(* CODESYS project AxisInterface0.0.1.32.library
   Company: Beckhoff Automation
   DefaultNamespace: BATW
   Version: 0.0.1.32
   Placeholder: AxisInterface
   Author: BATW
   Description: AxisInterface is used to control NC Axis
   Title: AxisInterface

Project tree, tasks and I/O mapping:
  libraries: BATW_Base, * (Beckhoff Automation); Common Behaviour Model, * (3S - Smart Software Solutions GmbH); Tc2_Math, * (Beckhoff Automation GmbH); Tc2_MC2, * (Beckhoff Automation GmbH); Tc2_MC2_Camming, * (Beckhoff Automation GmbH); Tc2_MC2_FlyingSaw, * (Beckhoff Automation GmbH); Tc2_Standard, * (Beckhoff Automation GmbH); Tc2_System, * (Beckhoff Automation GmbH); Tc2_Utilities, * (Beckhoff Automation GmbH); Tc3_JsonXml, * (Beckhoff Automation GmbH); Tc3_MC2_AdvancedHoming, * (Beckhoff Automation GmbH); Tc3_Module, * (Beckhoff Automation GmbH)
  AxisInterface/
    DUT/
      AdvancedHoming/
        data type E_HomingActionType
        data type ST_AdvancedHoming_Parameter
        data type ST_HomingCommand
        data type ST_HomingLimitation
        data type ST_PositionBiasParameter
        data type ST_StepFuncParameter
        data type ST_VelocityParameter
      Axis_Control/
        data type E_PositionType
        data type ST_AXIS_ADMINISTRATION
        data type ST_AXIS_CTRL
        data type ST_AXIS_POSITION
        data type ST_AXIS_SETUP_MODE
        data type ST_AXIS_SYNCHRONISATION
        data type ST_AXIS_SyncPhase
        data type ST_AXIS_SyncProfile
        data type ST_AXIS_SyncVel
        data type ST_AXIS_TORQUE
        data type ST_AXIS_VELOCITY
      Axis_Mode/
        data type E_AXIS_MODE
        data type E_HomingMode
        data type E_StartMode
        data type ST_AXIS_MODE_BITS
        data type U_AXIS_MODE
      Axis_Parameter/
        data type E_OS_Type
        data type ST_AXIS_Parameter
        data type ST_Backlash_Ctrl
        data type ST_Backlash_Status
        data type ST_PositionBias_Ctrl
      Axis_Status/
        data type ST_AXIS_ADMIN_STATUS
        data type ST_AXIS_DIAGNOSIS
        data type ST_AXIS_POS_STATUS
        data type ST_AXIS_SETUP_MODE_STATUS
        data type ST_AXIS_STATUS
        data type ST_AXIS_SYNC_STATUS
        data type ST_AXIS_VEL_STATUS
      CAM/
        data type E_CamID
        data type E_CamTableRef
        data type ST_CamTable
      data type E_AxisDirection
      data type E_MethodStatus_Basic
      data type E_NCI_Status
    GVL/
      global variables AxisInterface_Parameters
      global variables GVL_Motion
    LIB/
      AxisControl/
        program AxisInterface_Type01 [ST]
        function block FB_AdvancedHoming [ST]: M_ClearAllState, M_ClearSignal, M_SetBusy, M_SetDone, M_SetError, M_DogAbs, M_DogDetection, M_LimitDetection, M_LimitFind, M_MoveAbs, M_PulseDetection, M_PulseFind, M_AbortHoming, M_FinishHoming, M_HomeDirect, M_KeepPosBias, A_ActionTrigger, A_CyclicUpdate, M_CheckSignalConnected, M_SelectPreDefinedMode, M_SetUserDefinedMode
        function block FB_AxisControl [ST]: ClearAxisStatusBits, PowerOFF, PowerOn, ReleaseStopAxis, Reset, SetAxisDirction, StopAxis, A00_ModeAB, A01_ModeAH, A02_ModeAdvHoming, A02_ModeHoming, A03_ModePosAbs, A04_ModePosRel, A05_ModePosAdd, A06_ModeVel, A07_ModeSyncPhase, A08_ModeSyncVel, A09_ModeSyncCam, A10_ModeSyncProfile, A11_ModeTorque, A12_ModeFlexProfile, A13_ModeStopping, A14_ModeCoordinated, A15_ModeInterrupted, A16_ModeExternalFB, A17_ModeCyclicPosition, A18_ModeCyclicVelocity, A19_ModeCyclicTorque, A80_AxisParaHandle, A90_Cyclic, M_InitExtension
        function block MC_MoveAbsolute_Continue [ST]
        function block MC_MoveVelocity_Continue [ST]
  Basic Function/
    data type E_JsonHandlerAction
    function block FB_Json_Converter [ST]: JsonStrToObj, ObjToJsonStr
    function block FB_JsonHandler [ST]: CleanupAction, CyclicAction, StartAction, A_CyclicUpdate
  CorrugatedPrint/
    Feeder/
      function F_Poly7_MinTime [ST]
      function F_SolvePoly7Coefficients [ST]
      function block FB_CorrugatedLiftingCalculate [ST]: CleanupAction, CyclicAction, StartAction
      function block FB_CorrugatedWheelThreadCalculate [ST]: CyclicAction, StartAction
  program Main [ST]
*)

// AxisInterface/DUT/AdvancedHoming/E_HomingActionType
{attribute 'qualified_only'}
{attribute 'strict'}
(*
AdvancedHoming Function Type
1.Step Function / Finalizing Function
2.Ref Signal =Limit / Dog / Index
*)
TYPE E_HomingActionType :
(
	(*---Step Function---*)
	Limit_Detection 	:= 0,
	Limit_Abs			:= 1,
	Dog_Detection 		:= 4,
	Dog_Abs				:= 5,
	Index_Detection		:= 6,
	Index_Abs			:= 7,
	(*---Finalizing Function---*)
	HomeDirect			:= 8,
	FinishHoming		:= 9,
	(*---Parameter Setting Step---*)
	ParameterSetting	:=10,
	(*---Abs Motor move to Home---*)
	MoveAbs := 11
);
END_TYPE

// AxisInterface/DUT/AdvancedHoming/ST_AdvancedHoming_Parameter
TYPE ST_AdvancedHoming_Parameter :
STRUCT
	uiCommandNum			:UINT;					//Command List Number
	MovePara_Fast			:ST_VelocityParameter;	//High Speed
	MovePara_Slow			:ST_VelocityParameter;	//Low Speed
	bRefNegLimitSignal		:BOOL;					//Decide the LimitFind Ref Switch(Pos/Neg)
	stHomingCommand			:ARRAY[0..udiMAX_COMMAND_NUM-1] OF ST_HomingCommand;//Command List for Executing Adv Homing
END_STRUCT
END_TYPE

// AxisInterface/DUT/AdvancedHoming/ST_HomingCommand
TYPE ST_HomingCommand :
STRUCT
	eHome_ActionType		:E_HomingActionType;	//AdvancedHoming Function Type
	bSlowVelo				:BOOL;					//True, if Use Low Speed
	stStepFuncParameter		:ST_StepFuncParameter;	//AdvHoming Function Parameter
END_STRUCT
END_TYPE

// AxisInterface/DUT/AdvancedHoming/ST_HomingLimitation
TYPE ST_HomingLimitation :
STRUCT
	TimeLimit		:TIME:=T#0S;
	DistanceLimit	:LREAL:=0;
	TorqueLimit		:LREAL:=0;
END_STRUCT
END_TYPE

// AxisInterface/DUT/AdvancedHoming/ST_PositionBiasParameter
TYPE ST_PositionBiasParameter :
    STRUCT
        bSetPostionBias : BOOL;          //True, then Set Position Bias when Homing end.
        bModuloMode     : BOOL := FALSE; //True: Modulo Bias
    END_STRUCT
END_TYPE

// AxisInterface/DUT/AdvancedHoming/ST_StepFuncParameter
TYPE ST_StepFuncParameter :
STRUCT
	eHome_Direction			:MC_Home_Direction;		//Homing Starting Direction
	eSwitch_Mode			:MC_Switch_Mode;		//Switch Reaction Type
	MovePara				:ST_VelocityParameter;	//Movement Speed,this value should be set by Low/High Speed before Executing Homing Command List
	stHomingLimitation		:ST_HomingLimitation;	//Motion Limitation while searching
END_STRUCT
END_TYPE

// AxisInterface/DUT/AdvancedHoming/ST_VelocityParameter
TYPE ST_VelocityParameter :
STRUCT
	Velocity :LREAL;
	Acc :LREAL;
	Dec : LREAL;
	Jerk: LREAL;
END_STRUCT
END_TYPE

// AxisInterface/DUT/Axis_Control/E_PositionType
{attribute 'qualified_only'}
{attribute 'strict'}
TYPE E_PositionType :
(
	Linear := 0,
	Modulo
);
END_TYPE

// AxisInterface/DUT/Axis_Control/ST_AXIS_ADMINISTRATION
TYPE ST_AXIS_ADMINISTRATION :
    STRUCT
        Axis             : AXIS_REF;    // The reference to this Axis
        _OpMode          : U_AXIS_MODE; // Selection of the operating mode
        ClearError       : BOOL;        // Clear axis error with MC_Reset()
        StopDeceleration : LREAL :=100; // 
        PositionType     : E_PositionType;
        CommandDoneType  : BOOL; //True : real position arrived ;
        stBacklashCtrl   : ST_Backlash_Ctrl;

    END_STRUCT
END_TYPE

// AxisInterface/DUT/Axis_Control/ST_AXIS_CTRL
TYPE ST_AXIS_CTRL :
    STRUCT
        Admin      :ST_AXIS_ADMINISTRATION;  // Administration of the Axis
        PosMode    :ST_AXIS_POSITION;        // Operating mode positioning (absolute, rel, additive)
        VelMode    :ST_AXIS_VELOCITY;        // Operation mode velocity control
        SyncMode   :ST_AXIS_SYNCHRONISATION; // Operation mode synchronisation(phase, vel and cam)
        TorqueMode :ST_AXIS_TORQUE;          // Operation mode / force control
        SetupMode  :ST_AXIS_SETUP_MODE;      // Jog / Homing functionality
		//CoordinatedMode:ST_AXIS_Coordinated; // Operation mode Coordinated control (NCI)
    END_STRUCT
END_TYPE

// AxisInterface/DUT/Axis_Control/ST_AXIS_POSITION
// ST_AXIS_POSITION is a structure that contains the parameters needed when operating in position mode(ABS\REL).
TYPE
    ST_AXIS_POSITION :
    STRUCT
        Position : LREAL;      // The target position value in absolute mode.
        Distance : LREAL;      // The target distance value in relative mode.
        Velocity : LREAL;      // The velocity max value in the position motion.
        Acc : LREAL;           // The accelation max value in the position motion.
        Dec : LREAL;           // The decelation max value in the position motion.
        Jerk : LREAL;          // The jerk max value in the position motion.
        ContinueActive : BOOL; // True : Target command can be change while the motion still running.
    END_STRUCT
END_TYPE

// AxisInterface/DUT/Axis_Control/ST_AXIS_SETUP_MODE
TYPE ST_AXIS_SETUP_MODE :
STRUCT
	eHomingMode			:E_HomingMode;
	FastVelo			:ST_VelocityParameter;
	SlowVelo			:ST_VelocityParameter;
	FastLimitation		:ST_HomingLimitation;//Motion Limitation while Fast Searching
	SlowLimitation		:ST_HomingLimitation;//Motion Limitation while Slow Searching
	lrOffset			:LREAL;//Distance by which the axis moves away from the current position.
	lrSetPosition		:LREAL;//Position value to which the axis position is set to.
	stPosBiasParameter	:ST_PositionBiasParameter;
	
	bHomeSignal :BOOL;
	bPosLimitSignal :BOOL;
	bNegimitSignal :BOOL;
END_STRUCT
END_TYPE

// AxisInterface/DUT/Axis_Control/ST_AXIS_SYNCHRONISATION
TYPE ST_AXIS_SYNCHRONISATION :
STRUCT
	SyncVel :ST_AXIS_SyncVel;
	SyncPhase: ST_AXIS_SyncPhase;
	SyncProfile: ST_AXIS_SyncProfile;
END_STRUCT
END_TYPE

// AxisInterface/DUT/Axis_Control/ST_AXIS_SyncPhase
TYPE
    ST_AXIS_SyncPhase :
    STRUCT
        Master           : AXIS_REF;
        OutputRevolution : LREAL;
        InputRevolution  : UINT;
		MasterSyncPos : LREAL;
		SlaveSyncPos : LREAL;
		MaxAcceleration :LREAL;
		MaxDeceleration : LREAL;
		MaxJerk : LREAL;
		MaxVelocity :LREAL;
		
    //	StartMode        : E_StartMode;

    //  PhaseOffset      : LREAL;

    //  PhaseOffsetVel   : LREAL; // The velocity is used to phasing shift

    //  PhaseOffsetAcc   : LREAL; // The accelation is used to phasing shift

      SyncVelocity     : LREAL; // The velocity is the master axis and slave axis velocity diff in sync process

      SyncAcceleration : LREAL; // The acceleration is the master axis and slace axis acceleration diff in sync process
    END_STRUCT
END_TYPE

// AxisInterface/DUT/Axis_Control/ST_AXIS_SyncProfile
TYPE
    ST_AXIS_SyncProfile :
    STRUCT
        CamProfile    : ARRAY[1..4] OF MC_CAM_REF;
        MasterAxis    : AXIS_REF;
        ProfileNum    : UDINT; // Currently, only profiles 1 to 4 are supported (a total of 4 profiles).
        SyncType      : MC_StartMode;
        Periodic      : BOOL;
        MasterOffset  : LREAL; // Offset for the Master CamIn position, with the unit based on the NC configuration.
        SlaveOffset   : LREAL; // Offset for the Slace CamIn position, wtih the unit based on the NC configuration.
        MasterScaling : LREAL; // Master Axis position data scaling factor, init:1.0
        SlaveScaling  : LREAL; // Slave Axis position data scaling factor, init:1.0
    END_STRUCT
END_TYPE

// AxisInterface/DUT/Axis_Control/ST_AXIS_SyncVel
TYPE
    ST_AXIS_SyncVel :
    STRUCT
        OutputRevolution : LREAL;
        InputRevolution  : UINT;
        FineAdjust       : LREAL;
        Master           : AXIS_REF;
        Acceleration     : LREAL;
        Deceleration     : LREAL;
        Jerk             : LREAL;
    END_STRUCT
END_TYPE

// AxisInterface/DUT/Axis_Control/ST_AXIS_TORQUE
TYPE ST_AXIS_TORQUE :
STRUCT
END_STRUCT
END_TYPE

// AxisInterface/DUT/Axis_Control/ST_AXIS_VELOCITY
TYPE ST_AXIS_VELOCITY :
STRUCT
	Velocity :LREAL;
	Acc :LREAL;
	Dec : LREAL;
	Jerk: LREAL;
END_STRUCT
END_TYPE

// AxisInterface/DUT/Axis_Mode/E_AXIS_MODE
TYPE E_AXIS_MODE :
    (
        ModeAb             := 0,
        ModeAH             := 1,
        ModeHoming         := 2,
        ModePosAbs         := 4,
        ModePosRel         := 8,
        ModePosAdd         := 16,
        ModeVel            := 32,
        ModeSyncPhase      := 64,
        ModeSyncVel        := 128,
        ModeSyncCam        := 256,
        ModeSyncProfile    := 512,
        ModeTorque         := 1024,
        ModeFlexProfile    := 2048,
        ModeStopping       := 4096,
        ModeCoordinated    := 8192,
        ModeInterrupted    := 16384,
        ModeExternalFB     := 32768,
        ModeCyclicPosition := 65536,
        ModeCyclicVelocity := 131072,
        ModeCyclicTorque   := 262144
    )UDINT;
END_TYPE

// AxisInterface/DUT/Axis_Mode/E_HomingMode
{attribute 'qualified_only'}
{attribute 'strict'}
//CiA402 Homing Mode
(*-----------------

_03  					=> Mode Number
_Pos 					=> Start Direction
_LimitOutterLeftIndex 	=> Final target position
_withLimit				=> Action will reverse when meets limit

-----------------*)
TYPE E_HomingMode :
(
	notDefined									:=0,
                              	
	//Limit Switch plus Index           	
	_01_Neg_LimitOutterRightIndex				:=1,
	_02_Pos_LimitOutterLeftIndex 				:=2,
	
	//Single Transition Home Switch plus Index
	_03_Pos_HomeOutterLeftIndex					:=3,
	_04_Pos_HomeInnerLeftIndex					:=4,
	_05_Neg_HomeOutterRightIndex				:=5,
	_06_Neg_HomeInnerRightIndex					:=6,
	
	//Limited Range Home Switch, Limit Switched and Index
	_07_Pos_HomeOutterLeftIndex_withLimit		:=7,
	_08_Pos_HomeInnerLeftIndex_withLimit		:=8,
	_09_Pos_HomeInnerRightIndex_withLimit		:=9,
	_10_Pos_HomeOutterRightIndex_withLimit		:=10,
	_11_Neg_HomeOutterRightIndex_withLimit		:=11,
	_12_Neg_HomeInnerRightIndex_withLimit		:=12,
	_13_Neg_HomeInnerLeftIndex_withLimit		:=13,
	_14_Neg_HomeOutterLeftIndex_withLimit		:=14,
	
	//----------------------------//
	//Home on Limit Switch
	_17_Neg_LimitOutterRight				:=17,
	_18_Pos_LimitOutterLeft					:=18,
	
	//Single Transition Home Switch
	_19_Pos_HomeOutterLeft					:=19,
	_20_Pos_HomeInnerLeft					:=20,
	_21_Neg_HomeOutterRight					:=21,
	_22_Neg_HomeInnerRight					:=22,
	
	//Two Transition Home Switch and Limit Switches
	_23_Pos_HomeOutterLeft_withLimit		:=23,
	_24_Pos_HomeInnerLeft_withLimit			:=24,
	
	//Two Transition Home Switch, Limit Switches and Index
	_25_Pos_HomeInnerRight_withLimit		:=25,
	_26_Pos_HomeOutterRight_withLimit		:=26,
	_27_Neg_HomeOutterRight_withLimit		:=27,
	_28_Neg_HomeInnerRight_withLimit		:=28,
	_29_Neg_HomeInnerLeft_withLimit			:=29,
	_30_Neg_HomeOutterLeft_withLimit		:=30,

	//Index
	_33_Neg_Index			:=33,
	_34_Pos_Index			:=34,
	                                        	
	//Set to current position               	
	_35_CurrentPosition		:=35,
	
	// Absolute Motor move to home point
	_36_MoveToAbsHomePoint := 36
	//--------------Customized--------------//
	//_36_CurrentPosition_WithBias	:=36
	
	
	
);
END_TYPE

// AxisInterface/DUT/Axis_Mode/E_StartMode
{attribute 'qualified_only'}
{attribute 'strict'}
TYPE E_StartMode :
(
	Absolute := 0, // flying coupling with abs sync only first execution
	Relative :=1, // flying coupling with rel sync only first execution
	Absolute_Rampin, // flying coupling with abs sync every execution
	Relative_Rampin // flying coupling with rel sync ecery execution
);
END_TYPE

// AxisInterface/DUT/Axis_Mode/ST_AXIS_MODE_BITS
TYPE ST_AXIS_MODE_BITS :
    STRUCT
        ModeAH             :BIT;
        ModeHoming         :BIT;
        ModePosAbs         :BIT;
        ModePosRel         :BIT;
        ModePosAdd         :BIT;
        ModeVel            :BIT;
        ModeSyncPhase      :BIT;
        ModeSyncVel        :BIT;
        ModeSyncCam        :BIT;
        ModeSyncProfile    :BIT;
        ModeTorque         :BIT;
        ModeFlexProfile    :BIT;
        ModeStopping       :BIT;
        ModeCoordinated    :BIT;
        ModeInterrupted    :BIT;
        ModeExternalFB     :BIT;
        ModeCyclicPosition :BIT;
        ModeCyclicVelocity :BIT;
        ModeCyclicTorque   :BIT;
    END_STRUCT
END_TYPE

// AxisInterface/DUT/Axis_Mode/U_AXIS_MODE
TYPE U_AXIS_MODE :
UNION
	en : E_AXIS_MODE;
	b: ST_AXIS_MODE_BITS;
END_UNION
END_TYPE

// AxisInterface/DUT/Axis_Parameter/E_OS_Type
{attribute 'qualified_only'}
{attribute 'strict'}
TYPE E_OS_Type :
(
	WinCE 	:= 0,
	Windows := 1
);
END_TYPE

// AxisInterface/DUT/Axis_Parameter/ST_AXIS_Parameter
TYPE ST_AXIS_Parameter :
STRUCT
	(* -----Parameter----- *)
	(* Position Bias *)
	stPositionBias_Ctrl		:ST_PositionBias_Ctrl;
	
	(* Backlash *)
	stBacklash_Ctrl			:ST_Backlash_Ctrl;
	
END_STRUCT
END_TYPE

// AxisInterface/DUT/Axis_Parameter/ST_Backlash_Ctrl
TYPE ST_Backlash_Ctrl :
STRUCT
	bEnable		:BOOL;		//true, enable backlash compensation
	lrRamp		:LREAL:=1;	//Velocity limit for entered backlash compensation. [mm/s]
	lrBacklash	:LREAL:=0;	//Backlash Value
	bIsPosDir	:BOOL:=TRUE;//True, if Backlash compensation for Pos Direction
END_STRUCT
END_TYPE

// AxisInterface/DUT/Axis_Parameter/ST_Backlash_Status
TYPE ST_Backlash_Status :
STRUCT
	lrCurrentBacklash	:LREAL;//Current compensation value [mm].
	
	
END_STRUCT
END_TYPE

// AxisInterface/DUT/Axis_Parameter/ST_PositionBias_Ctrl
TYPE ST_PositionBias_Ctrl :
STRUCT
	lrPosBiasValue	:LREAL;//Position Bias Value 
	bSetPostionBias	:BOOL;//True, then Set Position Bias when Homing end.
	bModuloMode		:BOOL;//True=Modulo Bias
END_STRUCT
END_TYPE

// AxisInterface/DUT/Axis_Status/ST_AXIS_ADMIN_STATUS
TYPE
    ST_AXIS_ADMIN_STATUS :
    STRUCT
        Active             : BOOL;               // True: The drive is actived / PowerOn / Servo On
        CmdDone            : BOOL;               // Last motion command is finished
        _OpModeAck         : E_AXIS_MODE;        // acknowledge of the operation mode
        DriverAddress      : ST_DriveAddress;    // Read Driver Address
        stBacklash_Status  : ST_Backlash_Status; //Backlash Status
        ModeAb             : BIT;                // The axis is in Ab mode.
        ModeAH             : BIT;                // The axis is in AH mode.
        ModeHoming         : BIT;                // The axis is in homing mode.
        ModePosAbs         : BIT;                // The axis is in position absolute mode.
        ModePosRel         : BIT;                // This axis is in position relative mode.
        ModePosAdd         : BIT;                // This axis is in position additive mode.
        ModeVel            : BIT;                // This axis is in velocity control mode.
        ModeSyncPhase      : BIT;                // This axis is in synchronize phase mode.
        ModeSyncVel        : BIT;                // This axis is in synchronize velocity mode.
        ModeSyncCam        : BIT;                // This axis is in synchronize Cam mode.
        ModeSyncProfile    : BIT;                // This axis is in synchronize Cam Profile mode.
        ModeTorque         : BIT;                // This axis is in torque control mode.
        ModeFlexProfile    : BIT;                // This axis is in synchronize Cam-> FlexProfile mode.
        ModeStopping       : BIT;                // This axis is in stopping mode.
        ModeCoordinated    : BIT;                // This axis is in coordinated mode.
        ModeInterrupted    : BIT;                // This axis is in interrupted mode.
        ModeExternalFB     : BIT;                // This axis is using exeternal FB.
        ModeCyclicPosition : BIT;                // This axis is in cyclic Position control mode.
        ModeCyclicVelocity : BIT;                // This axis is in cyclic Velocity control mode.
        ModeCyclicTorque   : BIT;                // This axis is in cyclic torque control mode.
    END_STRUCT
END_TYPE

// AxisInterface/DUT/Axis_Status/ST_AXIS_DIAGNOSIS
TYPE ST_AXIS_DIAGNOSIS :
STRUCT
	Warning :BOOL := FALSE;
	Error : BOOL:=FALSE;
	ErrorID : UDINT;
	ErrorMsg : T_MaxString;
END_STRUCT
END_TYPE

// AxisInterface/DUT/Axis_Status/ST_AXIS_POS_STATUS
TYPE ST_AXIS_POS_STATUS :
STRUCT
END_STRUCT
END_TYPE

// AxisInterface/DUT/Axis_Status/ST_AXIS_SETUP_MODE_STATUS
TYPE ST_AXIS_SETUP_MODE_STATUS :
STRUCT
END_STRUCT
END_TYPE

// AxisInterface/DUT/Axis_Status/ST_AXIS_STATUS
TYPE ST_AXIS_STATUS :
    STRUCT
        Admin     :ST_AXIS_ADMIN_STATUS; 
        Diag      :ST_AXIS_DIAGNOSIS;
        PosMode   :ST_AXIS_POS_STATUS;
        VelMode   :ST_AXIS_VEL_STATUS;
        SyncMode  :ST_AXIS_SYNC_STATUS;
        SetupMode :ST_AXIS_SETUP_MODE_STATUS;
    END_STRUCT
END_TYPE

// AxisInterface/DUT/Axis_Status/ST_AXIS_SYNC_STATUS
TYPE
    ST_AXIS_SYNC_STATUS :
    STRUCT
        ModuleGap : LREAL;
    END_STRUCT
END_TYPE

// AxisInterface/DUT/Axis_Status/ST_AXIS_VEL_STATUS
TYPE ST_AXIS_VEL_STATUS :
STRUCT
END_STRUCT
END_TYPE

// AxisInterface/DUT/CAM/E_CamID
{attribute 'qualified_only'}
{attribute 'strict'}
TYPE E_CamID :
(
	Undefined := 0,
	Cam1 :=1,
	Cam2 :=2,
	Cam3 :=3,
	Cam4 :=4
)UDINT;
END_TYPE

// AxisInterface/DUT/CAM/E_CamTableRef
{attribute 'qualified_only'}
{attribute 'strict'}
TYPE
    E_CamTableRef :
    (
        Undefined := 0,
        CamTable_01 := 1,
        CamTable_02 := 2,
        CamTable_03 := 3,
        CamTable_04 := 4
    );
END_TYPE

// AxisInterface/DUT/CAM/ST_CamTable
TYPE
    ST_CamTable :
    STRUCT
        CamTable_01 : MC_CAM_REF;
        CamTable_02 : MC_CAM_REF;
        CamTable_03 : MC_CAM_REF;
        CamTable_04 : MC_CAM_REF;
    END_STRUCT
END_TYPE

// AxisInterface/DUT/E_AxisDirection
TYPE E_AxisDirection :
(
	Locked := 0,
	OnlyPositive,
	OnlyNegative,
	Both
)UINT;
END_TYPE

// AxisInterface/DUT/E_MethodStatus_Basic
// Declare the basic level that a method typically goes through, based on PLC Open OOP guidelines.
{attribute 'strict'}
TYPE E_MethodStatus_Basic :
(
	STATE_DORMANT := 0, // In dormant state, do nothing and just wait for the start command.
	STATE_EXECUTING, 	// In executing state, the state will do something that you coded
	STATE_ABORTING, 	// In aborting state, stop all ongoing commands.
	STATE_DONE, 		// In done state, waitting the reset command or execute signal off
	STATE_Aborted, 		// In aborted state, method is frozen wait reset command or execute signal off
	STATE_ERROR,		// In error state, method has been stopped and only can be restart by reset command or execute signal off 
	STATE_RESETTING    	// In resetting state, the state will revert the status to its initial values and clear any error signals.
)UDINT;
END_TYPE

// AxisInterface/DUT/E_NCI_Status
TYPE E_NCI_Status :
(
	NCI_INITFAILED := 0,
	NCI_IDLE,
	NCI_READY,
	NCI_STARTED,
	NCI_SCANNING,
	NCI_RUNNING,
	NCI_STAY_RUNNING,
	NCI_WRITETABLE,
	NCI_SEARCHLINE,
	NCI_END,
	NCI_SINGLESTOP,
	NCI_ABORTING,
	NCI_ABORTED,
	NCI_FAULT,
	NCI_RESET,
	NCI_STOP,
	NCI_WAITFUNC,
	NCI_FLUSHBUFFERS
)UDINT;
END_TYPE

// Basic Function/E_JsonHandlerAction
{attribute 'qualified_only'}
{attribute 'strict'}
TYPE E_JsonHandlerAction :
(
	READ 	:= 0,
	WRITE	:= 1
);
END_TYPE

// AxisInterface/GVL/AxisInterface_Parameters
VAR_GLOBAL CONSTANT
    uiMAX_AXIS_INDEX   		: UINT := 10;  // Maximum number of servos in the system.
    uiMAX_AXIS_NUMBER  		: UINT := 4;   // Actual number of servos in the system.
    udiMAX_COMMAND_NUM 		: UDINT := 10; //Maximum number of Advanced Homing command 
	eOsType			   		: E_OS_Type:=E_OS_Type.Windows;//OS Type,decide deafaut Axis Para file folder
	sAxisParaFolderPath  	: T_MaxString:='';//Axis Parameter File Folder ,example: 'C:\TwinCAT\3.1\Boot'
END_VAR

// AxisInterface/GVL/GVL_Motion
VAR_GLOBAL
    arAxisCtrl_gb     :ARRAY[1..uiMAX_AXIS_INDEX] OF ST_AXIS_CTRL;
    arAxisStatus_gb   :ARRAY[1..uiMAX_AXIS_INDEX] OF ST_AXIS_STATUS;
END_VAR
VAR_GLOBAL PERSISTENT
	arAxisPara_gb	  :ARRAY[1..uiMAX_AXIS_INDEX] OF ST_AXIS_Parameter;
	//arAxisBias_gb     		:ARRAY[1..uiMAX_AXIS_INDEX] OF LREAL;
END_VAR

// AxisInterface/LIB/AxisControl/AxisInterface_Type01
PROGRAM AxisInterface_Type01
VAR
    {attribute 'hide'}
    uiLoop :UINT; // For loop index
    {attribute 'hide'}
    fbAxis :ARRAY[1..uiMAX_AXIS_NUMBER] OF FB_AxisControl; // IMPLEMENTS axis control fb
	uiIndex : UINT;
	
	bDogSignal_Simu:BOOL;
	bPosLimitSiganl_Simu:BOOL;
	bNegLimitSignal_Simu:BOOL;
	
END_VAR

VAR CONSTANT
END_VAR

//============================================//
// Reflash Axis Interface					  //
//============================================//

FOR uiLoop := 1 TO uiMAX_AXIS_NUMBER DO
    fbAxis[uiLoop].M_InitExtension(uiLoop);
    //fbAxis[uiLoop]();
    fbAxis[uiLoop](HomeSensor := arAxisCtrl_gb[uiLoop].SetupMode.bHomeSignal,
                   PosLimit := arAxisCtrl_gb[uiLoop].SetupMode.bPosLimitSignal,
                   NegLimit := arAxisCtrl_gb[uiLoop].SetupMode.bNegimitSignal);
END_FOR

END_PROGRAM

// AxisInterface/LIB/AxisControl/FB_AxisControl
{attribute 'reflection'}
FUNCTION_BLOCK FB_AxisControl
VAR_INPUT
    HomeSensor : BOOL;
    PosLimit   : BOOL;
    NegLimit   : BOOL;

    {attribute 'hide'}
    bThirdPartyDrive : BOOL := TRUE;
END_VAR

VAR_OUTPUT
END_VAR

VAR
    // Control unit
    PowerControl          : Tc2_MC2.MC_Power; // MC_Power, Declare the use of a function block.
    ResetControl          : Tc2_MC2.MC_Reset; // MC_Reset, Declare the use of a function block.
    StopControl           : Tc2_MC2.MC_Stop; // MC_Stop, Declare the use of a function block.
    HaltControl           : Tc2_MC2.MC_Halt; // MC_Halt, Declare the use of a function block.
    JogControl            : Tc2_MC2.MC_Jog; // MC_Jog, Declare the use of a function block.
    HomingControl         : Tc2_MC2.MC_Home; // MC_Home, Declare the use of a function block.
    MoveAbsControl        : Tc2_MC2.MC_MoveAbsolute; // MC_MoveAbsolute, Declare the use of a function block.
    MoveRelControl        : Tc2_MC2.MC_MoveRelative; // MC_MoveRelative, Declare the use of a function block.
    MoveAddControl        : Tc2_MC2.MC_MoveAdditive; // MC_ModeAdditive, Declare the use of a function block.
    MoveModuleControl     : Tc2_MC2.MC_MoveModulo; // MC_MoveModule, Declare the use of a function block.
    MoveVelControl        : Tc2_MC2.MC_MoveVelocity; // MC_MoveVelocitu, Declare the use of a function block.
    MoveVelControl_Ext    : MC_MoveVelocity_Continue; // MC_MoveVelocity_Continue, Declare the use of a function block.
    MoveAbsolute_Ext      : MC_MoveAbsolute_Continue; // MC_MoveAbsolute_Continue, Declare the use of a function block.
    SyncVelControl        : MC_GearInVelo; // MC_GearInVelo, Declare the use of a function block.
    SyncPhaseControl      : MC_GearInPos; // MC_GearInPos, Declare the use of a function block.
    SetPositionControl    : MC_SetPosition; // MC_SetPositionControl, Declare the use of a function block.
    CamSelector           : MC_CamTableSelect; // MC_CamTableSelect, Declare the use of a function block.
    CamInControl          : MC_CamIn; // MC_CamIn, Declare the use of a function block.
    fbAdvancedHoming      : FB_AdvancedHoming; // FB_AdvancedHoming, Declare the use of a function block.
    fbBacklash            : MC_BacklashCompensation;
    PhasingAbsControl     : MC_PhasingAbsolute; // MC_PhasingAbsolute, Declare the use of a function block.
    PhasingRelControl     : MC_PhasingRelative; // MC_PhasingRelative, Declare the use of a function block.
    PhaseOffset_Abs       : LREAL;
    PhaseOffset_Rel       : LREAL;
    PhaseOffsetSuperInpos : MC_MoveSuperImposed;
    SuperInposMode        : E_SuperpositionMode;
    fbWriteNcPara         : MC_WriteParameterPersistent; //Read NC Parameter
    fbReadNcPara          : MC_ReadParameter; //Write NC Parameter
    fbWritePersistent     : FB_WritePersistentData;
    fbAxisParaHandler     : FB_JsonHandler;
    GearOutControl        : MC_GearOut;

    // Axis command 
    AxisPowerON       : BOOL; // True: set mc_power.enable = True
    AllowPositiveMove : BOOL; // True: Allow axis move to positive direction
    AllowNegativeMove : BOOL; // True: Allow axis move to Negative direction
    AxisStop          : BOOL; // True: Set mc_Stop.Execute = true
    AxisStop_Dec      : LREAL := 1000; // mc_Stop's deceleration
    AxisStop_Jerk     : LREAL := 10000; // mc_Stop's jerk
    AxisID            : UDINT;
    //-----Axis Parameter-----//
    //
    bInitializePosBiasDone : BOOL := FALSE;
    bReadAxisPara          : BOOL;
    sTempString            : STRING(255);
    sTempString2           : STRING(255);
    retryTimer             : TON;
    fbWritePersistentdata  : FB_WritePersistentData;
    lrNcCurrentBias        : LREAL;
    lrStoredBias           : LREAL;
    bAxisInitDone          : BOOL := FALSE;
    bAxisDoingInit         : BOOL := FALSE;
    uiAxisInitRetryCount   : UINT;

    //BackLash
    bBacklash_Enable   : BOOL; //true, enable backlash compensation
    lrBacklash_Ramp    : LREAL := 1; //Velocity limit for entered backlash compensation. [mm/s]
    lrBacklash_Value   : LREAL := 0; //Backlash Value
    bBacklash_IsPosDir : BOOL  := TRUE; //True, if Backlash compensation for Pos Direction

    // Cam Table
    CamProfileIndex : UDINT; // Cam Profile number (1~4)
    arCamID         : ARRAY[1..4] OF UDINT; // Store the actual CAM ID

    //A02 advance homing
    SetPosition_Execute       : BOOL;
    SetPosition_Position      : LREAL; // This value will be set to Absoulte position
    advHoming_eHomingMode     : E_HomingMode;
    advHoming_FastVelo        : ST_VelocityParameter;
    advHoming_SlowVelo        : ST_VelocityParameter;
    advHoming_lrOffset        : LREAL; //Distance by which the axis moves away from the current position.
    advHoming_lrSetPosition   : LREAL; //Position value to which the axis position is set to.
    advHoming_StartHoming     : BOOL;
    advHoming_AbortHoming     : BOOL;
    advHoming_ThirdPartyDrive : BOOL;
    {attribute 'is_connected' := 'HomeSensor'}
    advHoming_bDogConnected : BOOL;
    {attribute 'is_connected' := 'PosLimit'}
    advHoming_bPosLimitConnected : BOOL;
    {attribute 'is_connected' := 'NegLimit'}
    advHoming_bNegLimitConnected : BOOL;
    advHoming_PositionBiasPara   : ST_PositionBiasParameter;
	// A03
    PosAbsMode_Execute         : BOOL;
    PosAbsMode_Position        : LREAL;
    PosAbsMode_Velocity        : LREAL;
    PosAbsMode_Acc             : LREAL;
    PosAbsMode_Dec             : LREAL;
    PosAbsMode_Jerk            : LREAL;
    PosAbsMode_Exectue_Modulo  : BOOL;
    PosAbsMode_Position_Modulo : LREAL;
    PosAbsMode_Velocity_Modulo : LREAL;
    PosAbsMode_Acc_Modulo      : LREAL;
    PosAbsMode_Dec_Modulo      : LREAL;
    PosAbsMode_Jerk_Modulo     : LREAL;
	PosAbsMode_Direction : MC_Direction:=MC_Direction.MC_Shortest_Way;
	PosAbsMode_LastPosition : LREAL;
    //A04
    PosRelMode_Execute  : BOOL;
    PosRelMode_Distance : LREAL;
    PosRelMode_Velocity : LREAL;
    PosRelMode_Acc      : LREAL;
    PosRelMode_Dec      : LREAL;
    PosRelMode_Jerk     : LREAL;

    // A06
    VelMode_Velocity : LREAL := 0;
    VelMode_Acc      : LREAL := 10;
    VelMode_Dec      : LREAL := 10;
    VelMode_Jerk     : LREAL := 100;
    VelMode_Dir      : MC_Direction;
    VelMode_Execute  : BOOL;

    //A07 ModeSyncPhase
    SyncPhaseMode_Enable           : BOOL;
    SyncPhaseMode_Master           : REFERENCE TO AXIS_REF;
    SyncPhaseMode_RatioNumerator   : LREAL;
    SyncPhaseMode_RatioDenominator : UINT;
    SyncPhaseMode_MasterSyncPos    : LREAL := 0;
    SyncPhaseMode_SlaveSyncPos     : LREAL := 0;
    SyncPhaseMode_SyncMode         : ST_SyncMode;
    //SyncPhaseMode_MasterStartPos   : LREAL;
    SyncPhaseMode_MaxVelocity       : LREAL := 10;
    SyncPhaseMode_MaxAcc            : LREAL;
    SyncPhaseMode_MaxDec            : LREAL;
    SyncPhaseMode_MaxJerk           : LREAL;
    SyncPhaseMode_RealMasterPos     : LREAL;
    SyncPhaseMode_RealSlavePos      : LREAL;
    SyncPhaseMode_LastMasterSyncPos : LREAL;
    SyncPhaseMode_LastSlaveSyncPos  : LREAL;
    SyncPhaseMode_SyncVelocity      : LREAL;
    SyncPhaseMode_SyncAcceleration  : LREAL;
    //A08 ModeSyncVel
    SyncVelMode_Enable           : BOOL;
    SyncVelMode_Master           : REFERENCE TO AXIS_REF;
    SyncVelMode_GearRatio        : LREAL;
    SyncVelMode_RatioNumerator   : LREAL;
    SyncVelMode_RatioDenominator : UINT;
    SyncVelMode_SyncMode         : ST_SyncMode;
    SyncVelMode_FineAdjust       : LREAL;
    SyncVelMode_Acc              : LREAL;
    SyncVelMode_Dec              : LREAL;
    SyncVelMode_Jerk             : LREAL;

    //A10 ModeSyncProfile
    SyncProfileMode_Master        : REFERENCE TO AXIS_REF;
    SyncProfileMode_ProfileNum    : UDINT;
    SyncProfileMode_SyncType      : MC_StartMode;
    SyncProfileMode_MasterOffset  : LREAL;
    SyncProfileMode_SlaveOffset   : LREAL;
    SyncProfileMode_MasterScaling : LREAL := 1.0;
    SyncProfileMode_SlaveScaling  : LREAL := 1.0;
    SyncProfileMode_Periodic      : BOOL;
    SyncProfileMode_CamID         : MC_CAM_ID;
    SyncProfileOption             : ST_CamInOptions;

    //A17 ModeCyclicPosition
    PosCyclicAbsMode_Execute  : BOOL;
    PosCyclicAbsMode_Position : LREAL;
    PosCyclicAbsMode_Velocity : LREAL;
    PosCyclicAbsMode_Acc      : LREAL;
    PosCyclicAbsMode_Dec      : LREAL;
    PosCyclicAbsMode_Jerk     : LREAL;

    // Action state
    uiModeAb_State                      : UINT; // ModeAb's current state 
    uiModeAH_State                      : UINT; // ModeAH's current state
    uiModeHoming_State                  : UINT; // ModeHoming's current state
    uiModeCoordinatedState              : UINT; // ModeCoordinated current State
    uiModeVelState                      : UINT; // ModeVel's current state
    uiModePosAbsState                   : UINT; // ModePosAbs's current state
    uiModePosRelState                   : UINT; // ModePosRel's current state
    uiModeCyclicPosAbsState             : UINT; // ModePosAbs's current state
    uiModeSyncVelState                  : UINT; // ModeSyncVel's current state
    uiModeSyncPhaseState                : UINT; // ModeSyncPhase's current state
    uiModeSyncProfile                   : UINT; // ModeSyncProfile's current state
    uiModeFlexProfileState              : UINT; // ModeSyncFlexProfile current state
    LastOpMode                          : E_AXIS_MODE; // record last mode
    SyncPhaseMode_SlaveModuleTurns      : LREAL;
    SyncPhaseMode_SlaveModuleRemainder  : LREAL;
    SyncPhaseMode_MasterModuleTurns     : LREAL;
    SyncPhaseMode_MasterModuleRemainder : LREAL;
    SuperInposDistance                  : LREAL;
    AxesGap                             : LREAL;
    LastSuperInposDistance              : LREAL;

    // Read Axis Address
    fbReadAxisAddress : MC_ReadDriveAddress;
    AxesGap2          : LREAL;
    AxesGap3          : LREAL;
	ModuleGap: LREAL;
END_VAR

VAR
    {attribute 'no_copy'}
    AdminCtrl : REFERENCE TO ST_AXIS_ADMINISTRATION; // Reference to arAxisCtrl.admin
    {attribute 'no_copy'}
    PosModeCtrl : REFERENCE TO ST_AXIS_POSITION; // Reference to arAxisCtrl.PosMode
    {attribute 'no_copy'}
    VelModeCtrl : REFERENCE TO ST_AXIS_VELOCITY; // Reference to arAxisCtrl.VelMode
    {attribute 'no_copy'}
    SyncModeCtrl : REFERENCE TO ST_AXIS_SYNCHRONISATION; // Reference to arAxisCtrl SyncMode
    {attribute 'no_copy'}
    TorqueModeCtrl : REFERENCE TO ST_AXIS_TORQUE; // Reference to arAxisCtrl TorqueMode
    {attribute 'no_copy'}
    SetupModeCtrl : REFERENCE TO ST_AXIS_SETUP_MODE; // Reference to arAxisCtrl SetupMode
    {attribute 'no_copy'}
    AdminStatus : REFERENCE TO ST_AXIS_ADMIN_STATUS; // Reference to arAxisStat
    {attribute 'no_copy'}
    DiagStatus : REFERENCE TO ST_AXIS_DIAGNOSIS;
    {attribute 'no_copy'}
    PosModeStatus : REFERENCE TO ST_AXIS_POS_STATUS;
    {attribute 'no_copy'}
    VelModeStatus : REFERENCE TO ST_AXIS_VEL_STATUS;
    {attribute 'no_copy'}
    SyncModeStatus : REFERENCE TO ST_AXIS_SYNC_STATUS;
    {attribute 'no_copy'}
    SetupModeStatus : REFERENCE TO ST_AXIS_SETUP_MODE_STATUS;
    {attribute 'no_copy'}
    //refNcPositionBias : REFERENCE TO LREAL;//Reference to arAxisBias_gb
    {attribute 'no_copy'}
    refAxisPara : REFERENCE TO ST_AXIS_Parameter; //Reference to arAxisPara_gb
END_VAR

IF NOT __ISVALIDREF(AdminCtrl) THEN
    RETURN;
END_IF

// ----------------------------------------------- //
// ----------- Action ---------------------------- //
A00_ModeAB();
A01_ModeAH();
//A02_ModeHoming();
A02_ModeAdvHoming();
A03_ModePosAbs();
A04_ModePosRel();
A05_ModePosAdd();
A06_ModeVel();
A07_ModeSyncPhase();
A08_ModeSyncVel();
A09_ModeSyncCam();
A10_ModeSyncProfile();
A11_ModeTorque();
A12_ModeFlexProfile();
A13_ModeStopping();
A14_ModeCoordinated();
A15_ModeInterrupted();
A16_ModeExternalFB();
A17_ModeCyclicPosition();
A18_ModeCyclicVelocity();
A19_ModeCyclicTorque();

A90_Cyclic();

(* Axis Parameter Read/Write *)
A80_AxisParaHandle();

IF AdminCtrl.Axis.Status.Coupled THEN
    IF (SyncModeCtrl.SyncPhase.Master.NcToPlc.ModuloSetPos - AdminCtrl.Axis.NcToPlc.ModuloSetPos) >= 0 THEN
        ModuleGap := (SyncModeCtrl.SyncPhase.Master.NcToPlc.ModuloSetPos - AdminCtrl.Axis.NcToPlc.ModuloSetPos);
    ELSE
        ModuleGap := 360 + (SyncModeCtrl.SyncPhase.Master.NcToPlc.ModuloSetPos - AdminCtrl.Axis.NcToPlc.ModuloSetPos);
    END_IF
ELSE
    IF (SyncModeCtrl.SyncPhase.Master.NcToPlc.ModuloActPos - AdminCtrl.Axis.NcToPlc.ModuloActPos) >= 0 THEN
        ModuleGap := (SyncModeCtrl.SyncPhase.Master.NcToPlc.ModuloActPos - AdminCtrl.Axis.NcToPlc.ModuloActPos);
    ELSE
        ModuleGap := 360 + (SyncModeCtrl.SyncPhase.Master.NcToPlc.ModuloActPos - AdminCtrl.Axis.NcToPlc.ModuloActPos);
    END_IF
END_IF

SyncModeStatus.ModuleGap := ModuleGap;

METHOD PRIVATE ClearAxisStatusBits
VAR_INPUT
END_VAR
AdminStatus.ModeAb := FALSE;
AdminStatus.ModeAH := FALSE;
AdminStatus.ModeCoordinated := FALSE;
AdminStatus.ModeCyclicPosition := FALSE;
AdminStatus.ModeCyclicTorque := FALSE;
AdminStatus.ModeCyclicVelocity := FALSE;
AdminStatus.ModeExternalFB := FALSE;
AdminStatus.ModeFlexProfile := FALSE;
AdminStatus.ModeHoming := FALSE;
AdminStatus.ModeInterrupted := FALSE;
AdminStatus.ModePosAbs := FALSE;
AdminStatus.ModePosAdd := FALSE;
AdminStatus.ModePosRel := FALSE;
AdminStatus.ModeStopping := FALSE;
AdminStatus.ModeSyncCam := FALSE;
AdminStatus.ModeSyncPhase := FALSE;
AdminStatus.ModeSyncProfile := FALSE;
AdminStatus.ModeSyncVel := FALSE;
AdminStatus.ModeTorque := FALSE;
AdminStatus.ModeVel := FALSE;
END_METHOD

METHOD PRIVATE PowerOFF
VAR_INPUT
END_VAR
IF NOT PowerControl.Status THEN
    RETURN;
END_IF

AllowPositiveMove := FALSE;
AllowNegativeMove := FALSE;
AxisPowerON := FALSE;
END_METHOD

METHOD PRIVATE PowerOn
VAR_INPUT
    Direction :E_AxisDirection; // set the movable directions of the Axis.
END_VAR
VAR CONSTANT
	STATE_CHECK_AXISPOWER : UINT:=0;
	STATE_SET_POWER_PARA : UINT:=1;
END_VAR
IF PowerControl.Status THEN
	RETURN;
END_IF

SetAxisDirction(Direction:= Direction);

AxisPowerON := TRUE;
END_METHOD

METHOD ReleaseStopAxis :BOOL
VAR_INPUT
END_VAR
IF NOT AxisStop THEN
	RETURN;
END_IF

AxisStop := FALSE;

IF NOT StopControl.Active THEN
	IF Reset() THEN
		ReleaseStopAxis := TRUE;
	END_IF
END_IF
END_METHOD

METHOD Reset : BOOL
VAR_INPUT
END_VAR
IF NOT ResetControl.done THEN
    AdminCtrl.ClearError := TRUE;
END_IF
Reset := ResetControl.Done;
END_METHOD

METHOD PRIVATE SetAxisDirction
VAR_INPUT
	Direction : E_AxisDirection; // select axis direction
END_VAR
CASE Direction OF
	E_AxisDirection.Locked:
		AllowPositiveMove := FALSE;
		AllowNegativeMove := FALSE;
	E_AxisDirection.OnlyPositive:
		AllowPositiveMove := TRUE;
		AllowNegativeMove := FALSE;
	E_AxisDirection.OnlyNegative:
		AllowPositiveMove := FALSE;
		AllowNegativeMove := TRUE;
	E_AxisDirection.Both:
		AllowPositiveMove := TRUE;
		AllowNegativeMove := TRUE;
END_CASE
END_METHOD

METHOD StopAxis
VAR_INPUT
    StopDeceleration :LREAL := 1000;
    StopJerk         :LREAL := 10000;
END_VAR
IF (AdminCtrl.Axis.Status.StandStill AND AdminCtrl.Axis.Status.NotMoving) THEN
    RETURN;
END_IF

AxisStop_Dec  := StopDeceleration;
AxisStop_Jerk := StopJerk;
AxisStop      := TRUE;
END_METHOD

ACTION A00_ModeAB:
IF NOT __ISVALIDREF(AdminCtrl) THEN
    RETURN;
END_IF

IF AdminCtrl._OpMode.en <> ModeAb THEN
    HaltControl.Execute := FALSE;
    RETURN;
ELSIF AdminCtrl._OpMode.en <> LastOpMode THEN
    uiModeAb_State := 0;
    LastOpMode := AdminCtrl._OpMode.en;
END_IF

CASE uiModeAb_State of
    0:
        // Check Axis Status
        AdminStatus.CmdDone := FALSE;
        ClearAxisStatusBits();

        IF AdminCtrl.Axis.Status.Disabled AND NOT AxisPowerON THEN
            uiModeAb_State := 2000;
        ELSIF AdminCtrl.Axis.Status.Disabled AND AxisPowerON THEN
            AxisPowerON := FALSE;
            uiModeAb_State := 2000;
        ELSIF AdminCtrl.Axis.Status.Moving  OR AdminCtrl.Axis.Status.Coupled THEN
            uiModeAb_State := 100;
        END_IF
    100:

        VelMode_Execute := FALSE;
        HaltControl.Jerk := 1000;
        HaltControl.Deceleration := AdminCtrl.StopDeceleration;
        HaltControl.Execute := TRUE;
        uiModeAb_State := 200;
    200:
        IF HaltControl.Done THEN
            HaltControl.Execute := FALSE;
            uiModeAb_State := 300;
        END_IF
	300:
        IF AdminCtrl.Axis.Status.Coupled THEN
            GearOutControl.Execute := TRUE;
            uiModeAb_State := 400;
        ELSE
            uiModeAb_State := 1000;
        END_IF
    400:
        IF GearOutControl.Done THEN
            uiModeAb_State := 1000;
        END_IF
    1000:
        // Set MC_Power disable
        PowerOFF();
        ReleaseStopAxis();

        IF AdminCtrl.Axis.Status.Disabled THEN
            uiModeAb_State := 2000;
        END_IF
    (*==========Initialize==========*)
    2000:
        IF NOT bAxisInitDone THEN
            (* Wait Read Var Done*)
            IF bInitializePosBiasDone THEN
                //Get Stored Bias Value
                //lrStoredBias	:= refNcPositionBias;
                lrStoredBias := refAxisPara.stPositionBias_Ctrl.lrPosBiasValue;

                //Write to NC
                fbWriteNcPara.ParameterNumber := MC_AxisParameter.AxisEncoderOffset; //Position Bias
                fbWriteNcPara.Value := lrStoredBias;
                fbWriteNcPara.Execute := TRUE;

                uiModeAb_State := 2010;

            END_IF
        ELSE
            uiModeAb_State := 9000;
        END_IF
    2010: //Wait Done

        IF fbWriteNcPara.Done THEN
            fbWriteNcPara.Execute := FALSE;

            bAxisInitDone := TRUE;

            uiModeAb_State := 9000;

        ELSIF fbWriteNcPara.Error THEN
            //uiErrorId:=9930;
        END_IF
    (*-----------------------------*)
    9000:
        // Setting Axis Status
        AdminStatus.CmdDone := TRUE;
        AdminStatus.ModeAb := TRUE;
        AdminStatus._OpModeAck := ModeAb;

    10000:
END_CASE
END_ACTION

ACTION A01_ModeAH:
IF NOT __ISVALIDREF(AdminCtrl) THEN
	RETURN;
END_IF

IF AdminCtrl._OpMode.en <> ModeAH THEN
	RETURN;
ELSIF AdminCtrl._OpMode.en <> LastOpMode THEN
	uiModeAH_State := 0;
	LastOpMode := AdminCtrl._OpMode.en;
END_IF

CASE uiModeAH_State OF
	0:
		AdminStatus.CmdDone := FALSE;
		AdminStatus.ModeAH := TRUE;
		AdminStatus._OpModeAck := ModeAH;
        ClearAxisStatusBits();
		uiModeAH_State := 10;
	10:
		
		// Check Axis Status
		IF AdminCtrl.Axis.Status.Disabled AND NOT AxisPowerON THEN
			uiModeAH_State := 100;
		ELSIF AdminCtrl.Axis.Status.Disabled AND AxisPowerON THEN
			PowerOFF();
			IF  NOT AdminStatus.Active THEN
				uiModeAH_State := 200;
			END_IF
		ELSE
			uiModeAH_State := 200;
		END_IF
	100:
		// Power off -> Power On
		PowerOn(Direction:= E_AxisDirection.Both);
		IF PowerControl.Status THEN
			uiModeAH_State := 200;
		END_IF
	200:
		IF AdminCtrl.Axis.Status.StandStill AND AdminCtrl.Axis.Status.NotMoving THEN
			uiModeAH_State := 9000;
		ELSE
			uiModeAH_State := 300;
		END_IF
	300:
		// Stop Axis
		AxisStop := TRUE;
		AxisStop_Dec := AdminCtrl.StopDeceleration;
		IF StopControl.Done THEN
			uiModeAH_State := 400;
		END_IF
	400:
		AxisStop := FALSE;
		AdminCtrl.ClearError := TRUE;
		IF ResetControl.Done THEN
			uiModeAH_State := 500;
		END_IF
	500:
		AdminCtrl.ClearError := FALSE;
		ClearAxisStatusBits();
		uiModeAH_State := 8000;
		
	(*---Set Axis ---*)
	8000://Set Backlash
		
		IF AdminCtrl.stBacklashCtrl.bEnable THEN
			
			bBacklash_Enable	:=TRUE;
			lrBacklash_Ramp		:=AdminCtrl.stBacklashCtrl.lrRamp;
			lrBacklash_Value	:=AdminCtrl.stBacklashCtrl.lrBacklash;
			bBacklash_IsPosDir	:=AdminCtrl.stBacklashCtrl.bIsPosDir;
			
			uiModeAH_State:=8100;
		ELSE//Backlash not Enabled
			uiModeAH_State:=9000;
		END_IF
		
	8100:
		IF fbBacklash.Enabled THEN
			uiModeAH_State:=9000;
		END_IF
	9000:
	
		// Setting Axis Status
		AdminStatus.CmdDone := TRUE;
		uiModeAH_State := 10000;

	10000:
		// Wait Command
END_CASE
END_ACTION

ACTION A02_ModeAdvHoming:
IF NOT __ISVALIDREF(AdminCtrl) THEN
    RETURN;
END_IF

IF AdminCtrl._OpMode.en <> ModeHoming THEN
    advHoming_AbortHoming := FALSE;
	advHoming_StartHoming := FALSE;
    RETURN;
ELSIF AdminCtrl._OpMode.en <> LastOpMode THEN
    uiModeHoming_State := 0;
    LastOpMode     := AdminCtrl._OpMode.en;
END_IF


////fbAdvancedHoming.refNcPositionBias REF= THIS^.refNcPositionBias;
//fbAdvancedHoming.refAxisPara REF= THIS^.refAxisPara;

CASE uiModeHoming_State OF
    0:
        AdminStatus.CmdDone    := FALSE;
        AdminStatus.ModeHoming := TRUE;
        AdminStatus._OpModeAck := ModeHoming;
        ClearAxisStatusBits();
        uiModeHoming_State := 10;
    10:
        // Check Axis Status
        IF AdminCtrl.Axis.Status.Disabled THEN
            uiModeHoming_State := 100;
        ELSE
            uiModeHoming_State := 200;
        END_IF
    100:
        // Power off -> Power On
        PowerOn(Direction := E_AxisDirection.Both);

        IF PowerControl.Status THEN
            uiModeHoming_State := 200;
        END_IF
    200:
        IF AdminCtrl.Axis.Status.StandStill AND AdminCtrl.Axis.Status.NotMoving THEN
            uiModeHoming_State := 600;
        ELSE
            uiModeHoming_State := 300;
        END_IF
    300:
        // Stop Axis
        AxisStop     := TRUE;
        AxisStop_Dec := AdminCtrl.StopDeceleration;

        IF StopControl.Done THEN
            uiModeHoming_State := 400;
        END_IF
    400:
        AxisStop             := FALSE;
        AdminCtrl.ClearError := TRUE;

        IF ResetControl.Done THEN
            uiModeAH_State := 500;
        END_IF
    500:
        AdminCtrl.ClearError := FALSE;
        uiModeHoming_State   := 600;
    600: // Select homing mode

		advHoming_FastVelo			:=SetupModeCtrl.FastVelo;
		advHoming_SlowVelo			:=SetupModeCtrl.SlowVelo;
		advHoming_lrOffset			:=SetupModeCtrl.lrOffset;
		advHoming_lrSetPosition		:=SetupModeCtrl.lrSetPosition;
	
		advHoming_eHomingMode		:=SetupModeCtrl.eHomingMode;
		advHoming_ThirdPartyDrive	:=THIS^.bThirdPartyDrive;
		
		advHoming_PositionBiasPara	:=SetupModeCtrl.stPosBiasParameter;
		
		//Set Mode
		fbAdvancedHoming.M_SelectPreDefinedMode(advHoming_eHomingMode,advHoming_PositionBiasPara.bSetPostionBias);
		
		uiModeHoming_State := 700;
		
    700:
        advHoming_StartHoming  := TRUE;
		
        uiModeHoming_State   := 9000;
    9000:
		IF fbAdvancedHoming.Done THEN
			
			//Save Position Bias
			
			////refNcPositionBias								:=	fbAdvancedHoming.lrPosBiasValue;
			refAxisPara.stPositionBias_Ctrl.lrPosBiasValue	:=	fbAdvancedHoming.lrPosBiasValue;
			
			uiModeHoming_State := 9100;
		END_IF
	(* ---Save Parameter--- *)
	9100://Write Persistent
	
		fbWritePersistent.PORT	:= 851;
		fbWritePersistent.START	:= TRUE;
		
		IF NOT fbWritePersistent.BUSY AND NOT fbWritePersistent.ERR THEN
			fbWritePersistent.START	:= FALSE;
			uiModeHoming_State := 9200;
		ELSIF fbWritePersistent.ERR THEN
			;
		END_IF
	9200:(* Write File *)

		(* User defined path exists *)
		IF sAxisParaFolderPath <> '' THEN
			sTempString:=CONCAT(sAxisParaFolderPath,'\AxisParameter_');
			sTempString2:=CONCAT(TO_STRING(AdminCtrl.Axis.NcToPlc.AxisId),'.json');
			fbAxisParaHandler.sFilePath := CONCAT(sTempString, sTempString2);
		ELSE
			(* Default File path *)
			IF eOsType = E_OS_Type.WinCE THEN
				sTempString	:='\Hard Disk\TwinCAT\3.1\Boot\AxisParameter_';
				sTempString2:=CONCAT(TO_STRING(AdminCtrl.Axis.NcToPlc.AxisId),'.json');
				fbAxisParaHandler.sFilePath := CONCAT(sTempString, sTempString2);
			ELSIF eOsType = E_OS_Type.Windows  THEN
				sTempString	:='C:\TwinCAT\3.1\Boot\AxisParameter_';
				sTempString2:=CONCAT(TO_STRING(AdminCtrl.Axis.NcToPlc.AxisId),'.json');
				fbAxisParaHandler.sFilePath := CONCAT(sTempString, sTempString2);
			END_IF
		END_IF
		
		fbAxisParaHandler.eAction 	:= E_JsonHandlerAction.WRITE;
		fbAxisParaHandler.pData 	:= ADR(refAxisPara);
		fbAxisParaHandler.nData 	:= SIZEOF(refAxisPara);
		
		fbAxisParaHandler.xExecute	:=TRUE;
		
		IF fbAxisParaHandler.xDone THEN
			fbAxisParaHandler.xExecute:=FALSE;
			uiModeHoming_State := 10000;
		END_IF
		
    10000:
		advHoming_StartHoming:=FALSE;
        AdminStatus.CmdDone := TRUE;
		uiModeHoming_State := 11000;
	11000:
		// Wait command
END_CASE
END_ACTION

ACTION A02_ModeHoming:
IF NOT __ISVALIDREF(AdminCtrl) THEN
    RETURN;
END_IF

IF AdminCtrl._OpMode.en <> ModeHoming THEN
    SetPosition_Execute := FALSE;
    RETURN;
ELSIF AdminCtrl._OpMode.en <> LastOpMode THEN
    uiModeHoming_State := 0;
    LastOpMode     := AdminCtrl._OpMode.en;
END_IF

CASE uiModeHoming_State OF
    0:
        AdminStatus.CmdDone    := FALSE;
        AdminStatus.ModeHoming := TRUE;
        AdminStatus._OpModeAck := ModeHoming;
        ClearAxisStatusBits();
        uiModeHoming_State := 10;
    10:
        // Check Axis Status
        IF AdminCtrl.Axis.Status.Disabled THEN
            uiModeHoming_State := 100;
        ELSE
            uiModeHoming_State := 200;
        END_IF
    100:
        // Power off -> Power On
        PowerOn(Direction := E_AxisDirection.Both);

        IF PowerControl.Status THEN
            uiModeHoming_State := 200;
        END_IF
    200:
        IF AdminCtrl.Axis.Status.StandStill AND AdminCtrl.Axis.Status.NotMoving THEN
            uiModeHoming_State := 600;
        ELSE
            uiModeHoming_State := 300;
        END_IF
    300:
        // Stop Axis
        AxisStop     := TRUE;
        AxisStop_Dec := AdminCtrl.StopDeceleration;

        IF StopControl.Done THEN
            uiModeHoming_State := 400;
        END_IF
    400:
        AxisStop             := FALSE;
        AdminCtrl.ClearError := TRUE;

        IF ResetControl.Done THEN
            uiModeAH_State := 500;
        END_IF
    500:
        AdminCtrl.ClearError := FALSE;
        uiModeHoming_State   := 600;
    600: // Select homing mode
        IF SetupModeCtrl.eHomingMode = E_HomingMode._35_CurrentPosition THEN
            uiModeHoming_State := 700;
        END_IF
    700:
        SetPosition_Execute  := TRUE;
        SetPosition_Position := SetupModeCtrl.lrSetPosition;
        uiModeHoming_State   := 9000;
    9000:
		IF SetPositionControl.Done THEN
			uiModeHoming_State := 10000;
		END_IF
    10000:
        AdminStatus.CmdDone := TRUE;
		uiModeHoming_State := 11000;
	11000:
		// Wait command
END_CASE
END_ACTION

ACTION A03_ModePosAbs:
IF NOT __ISVALIDREF(AdminCtrl) THEN
    RETURN;
END_IF

IF AdminCtrl._OpMode.en <> ModePosAbs THEN
    PosAbsMode_Execute := FALSE;
    PosAbsMode_Exectue_Modulo := FALSE;
    RETURN;
ELSIF AdminCtrl._OpMode.en <> LastOpMode THEN
    uiModePosAbsState := 0;
    LastOpMode := AdminCtrl._OpMode.en;
END_IF

CASE uiModePosAbsState OF
    0:
        AdminStatus.CmdDone := FALSE;
        ClearAxisStatusBits();
        uiModePosAbsState := 10;
    10:
        AdminStatus.ModePosAbs := TRUE;
        AdminStatus._OpModeAck := ModePosAbs;
        PosAbsMode_Execute := FALSE;

        IF AdminCtrl.Axis.Status.Disabled THEN
            uiModePosAbsState := 100;
        ELSE
            IF AdminCtrl.PositionType = E_PositionType.Linear THEN
                uiModePosAbsState := 200;
            ELSIF AdminCtrl.PositionType = E_PositionType.Modulo THEN
                uiModePosAbsState := 300;
            END_IF
        END_IF
    100:
        // Power off -> Power On
        PowerOn(Direction := E_AxisDirection.Both);

        IF PowerControl.Status THEN
            IF AdminCtrl.PositionType = E_PositionType.Linear THEN
                uiModePosAbsState := 200;
            ELSIF AdminCtrl.PositionType = E_PositionType.Modulo THEN
                uiModePosAbsState := 300;
            END_IF
        END_IF
    200:
        PosAbsMode_Position := PosModeCtrl.Position;
        PosAbsMode_Velocity := PosModeCtrl.Velocity;
        PosAbsMode_Acc := PosModeCtrl.Acc;
        PosAbsMode_Dec := PosModeCtrl.Dec;
        PosAbsMode_Jerk := PosModeCtrl.Jerk;
        PosAbsMode_Execute := TRUE;

        //        uiModePosAbsState   := 9000;
        IF MoveAbsolute_Ext.Done THEN
            AdminStatus.CmdDone := TRUE;
        ELSE
            AdminStatus.CmdDone := FALSE;
        END_IF

        IF MoveAbsolute_Ext.CommandAborted OR MoveAbsolute_Ext.Error THEN
            ;
        END_IF
    300:
        PosAbsMode_Position_Modulo := PosModeCtrl.Position;
        PosAbsMode_Velocity_Modulo := PosModeCtrl.Velocity;
        PosAbsMode_Acc_Modulo := PosModeCtrl.Acc;
        PosAbsMode_Dec_Modulo := PosModeCtrl.Dec;
        PosAbsMode_Jerk_Modulo := PosModeCtrl.Jerk;
        PosAbsMode_Direction := MC_Direction.MC_Shortest_Way;
        PosAbsMode_Exectue_Modulo := TRUE;
		uiModePosAbsState := 400;
	400:
		
        IF MoveModuleControl.Done THEN
            AdminStatus.CmdDone := TRUE;
			PosAbsMode_LastPosition := PosModeCtrl.Position;
			PosAbsMode_Exectue_Modulo := FALSE;
			uiModePosAbsState := 500;
        ELSE
            AdminStatus.CmdDone := FALSE;
        END_IF

        IF MoveModuleControl.CommandAborted OR MoveModuleControl.Error THEN
            ;
        END_IF
	500:	
		IF PosAbsMode_LastPosition <> PosModeCtrl.Position THEN
			PosAbsMode_Exectue_Modulo := FALSE;
			AdminStatus.CmdDone := FALSE;
			uiModePosAbsState := 300;
		END_IF
		
END_CASE
END_ACTION

ACTION A04_ModePosRel:
IF NOT __ISVALIDREF(AdminCtrl) THEN
    RETURN;
END_IF

IF AdminCtrl._OpMode.en <> ModePosRel THEN
    RETURN;
ELSIF AdminCtrl._OpMode.en <> LastOpMode THEN
    uiModePosAbsState := 0;
    LastOpMode     := AdminCtrl._OpMode.en;
END_IF

CASE uiModePosRelState OF
	0:
		AdminStatus.CmdDone := FALSE;
        ClearAxisStatusBits();
		uiModePosRelState := 10;	
	10:
		AdminStatus.ModePosAbs := TRUE;
		AdminStatus._OpModeAck := ModePosRel;
		PosRelMode_Execute     := FALSE;
		
		IF AdminCtrl.Axis.Status.Disabled THEN
            uiModePosRelState := 100;
        ELSE
            uiModePosRelState := 200;
        END_IF	
	100:
		// Power off -> Power On
        PowerOn(Direction := E_AxisDirection.Both);

        IF PowerControl.Status THEN
            uiModePosRelState := 200;
        END_IF
	200:
		PosRelMode_Distance := PosModeCtrl.Distance;
        PosRelMode_Velocity := PosModeCtrl.Velocity;
        PosRelMode_Acc      := PosModeCtrl.Acc;
        PosRelMode_Dec      := PosModeCtrl.Dec;
        PosRelMode_Jerk     := PosModeCtrl.Jerk;
        PosRelMode_Execute  := TRUE;
        uiModePosRelState   := 9000;
	9000:
		IF MoveRelControl.Done THEN
            AdminStatus.CmdDone := TRUE;
            uiModePosRelState := 10000;
        ELSIF MoveRelControl.CommandAborted OR MoveRelControl.Error THEN
            uiModePosRelState := 20000;
        END_IF;
	10000:
		// Wait Command
		IF PosModeCtrl.Distance <> PosModeCtrl.Distance THEN
			PosRelMode_Execute := FALSE;
            AdminStatus.CmdDone := FALSE;
			uiModePosRelState := 200;
		END_IF
END_CASE
END_ACTION

ACTION A05_ModePosAdd:

END_ACTION

ACTION A06_ModeVel:
IF NOT __ISVALIDREF(AdminCtrl) THEN
    RETURN;
END_IF

IF AdminCtrl._OpMode.en <> ModeVel THEN
	VelMode_Execute := FALSE;
    RETURN;
ELSIF AdminCtrl._OpMode.en <> LastOpMode THEN
    uiModeVelState := 0;
    LastOpMode     := AdminCtrl._OpMode.en;
END_IF

CASE uiModeVelState OF
    0:
        AdminStatus.CmdDone := FALSE;
		ClearAxisStatusBits();
		uiModeVelState      := 10;
	10:
        AdminStatus.ModeVel := TRUE;
		AdminStatus._OpModeAck := ModeVel;
        VelMode_Execute     := FALSE;
		ReleaseStopAxis();
        // Check Axis Status
		IF AdminCtrl.Axis.Status.Disabled AND NOT AxisPowerON THEN
			uiModeVelState := 100;
		ELSIF AdminCtrl.Axis.Status.Disabled AND AxisPowerON THEN
			PowerOFF();
			IF  NOT AdminStatus.Active THEN
				uiModeVelState := 200;
			END_IF
		ELSE
			uiModeVelState := 200;
		END_IF
    100:
        // Power off -> Power On
        PowerOn(Direction := E_AxisDirection.Both);

        IF AdminCtrl.Axis.Status.ControlLoopClosed THEN
            uiModeVelState := 200;
        END_IF
//	110:
//		IF AdminCtrl.
    200:
        VelMode_Acc      := VelModeCtrl.Acc;
        VelMode_Dec      := VelModeCtrl.Dec;
        VelMode_Jerk     := VelModeCtrl.Jerk;

		VelMode_Velocity := VelModeCtrl.Velocity;
        IF VelModeCtrl.Velocity > 0 THEN
            VelMode_Dir := MC_Direction.MC_Positive_Direction;
        ELSIF VelModeCtrl.Velocity < 0 THEN
            VelMode_Dir := MC_Direction.MC_Negative_Direction;
        END_IF
		VelMode_Execute  := TRUE;
		
		AdminStatus.CmdDone := MoveVelControl_Ext.InVeloctiy;
END_CASE
END_ACTION

ACTION A07_ModeSyncPhase:
IF NOT __ISVALIDREF(AdminCtrl) THEN
    RETURN;
END_IF

IF AdminCtrl._OpMode.en <> ModeSyncPhase THEN
    SyncPhaseMode_Enable := FALSE;
    PhasingAbsControl.Execute := FALSE;
    PhaseOffsetSuperInpos.Execute := FALSE;
    RETURN;
ELSIF AdminCtrl._OpMode.en <> LastOpMode THEN
    uiModeSyncPhaseState := 0;
    LastOpMode := AdminCtrl._OpMode.en;
END_IF

// Module Master axis and Slave axis ActPos
SyncPhaseMode_SlaveModuleTurns := TRUNC(AdminCtrl.Axis.NcToPlc.ActPos / 360.0);

//SyncPhaseMode_SlaveModuleRemainder  := ABS(LMOD(AdminCtrl.Axis.NcToPlc.ActPos, 360));
SyncPhaseMode_SlaveModuleRemainder := AdminCtrl.Axis.NcToPlc.ModuloActPos;
SyncPhaseMode_MasterModuleTurns := TRUNC(SyncModeCtrl.SyncPhase.Master.NcToPlc.ActPos / 360.0);

//SyncPhaseMode_MasterModuleRemainder := ABS(LMOD(SyncModeCtrl.SyncPhase.Master.NcToPlc.ActPos, 360));
SyncPhaseMode_MasterModuleRemainder := SyncModeCtrl.SyncPhase.Master.NcToPlc.ModuloActPos;
//IF (SyncModeCtrl.SyncPhase.Master.NcToPlc.ModuloSetPos - AdminCtrl.Axis.NcToPlc.ModuloSetPos) >=0 THEN
//	ModuleGap := (SyncModeCtrl.SyncPhase.Master.NcToPlc.ModuloSetPos - AdminCtrl.Axis.NcToPlc.ModuloSetPos);
//ELSE
//	ModuleGap := 360 + (SyncModeCtrl.SyncPhase.Master.NcToPlc.ModuloSetPos - AdminCtrl.Axis.NcToPlc.ModuloSetPos);
//END_IF

CASE uiModeSyncPhaseState OF
    0:
        AdminStatus.CmdDone := FALSE;
        ClearAxisStatusBits();
        uiModeSyncPhaseState := 10;
    10:
        AdminStatus.ModeSyncVel := TRUE;
        AdminStatus._OpModeAck := ModeSyncPhase;
        SyncVelMode_Enable := TRUE;

        IF AdminCtrl.Axis.Status.Disabled THEN
            uiModeSyncPhaseState := 100;
        ELSE
            uiModeSyncPhaseState := 200;
        END_IF
    100:
        // Power off -> Power On
        PowerOn(Direction := E_AxisDirection.Both);

        IF PowerControl.Status THEN
            uiModeSyncPhaseState := 200;
        END_IF
    200:
        IF AdminCtrl.PositionType = E_PositionType.Linear THEN
            uiModeSyncPhaseState := 300;
        ELSIF AdminCtrl.PositionType = E_PositionType.Modulo THEN
            uiModeSyncPhaseState := 400;
        END_IF
    300:
        IF AdminCtrl.PositionType = E_PositionType.Modulo THEN
            SyncPhaseMode_RealMasterPos := SyncModeCtrl.SyncPhase.MasterSyncPos + SyncModeCtrl.SyncPhase.Master.NcToPlc.ActPos + 10;
            SyncPhaseMode_RealSlavePos := SyncModeCtrl.SyncPhase.SlaveSyncPos + AdminCtrl.Axis.NcToPlc.ActPos;
        ELSIF AdminCtrl.PositionType = E_PositionType.Linear THEN
            //SyncPhaseMode_RealMasterPos
        END_IF

        SyncPhaseMode_Master REF= SyncModeCtrl.SyncPhase.Master;
        SyncPhaseMode_MasterSyncPos := SyncPhaseMode_RealMasterPos;
        SyncPhaseMode_SlaveSyncPos := SyncPhaseMode_RealSlavePos;
        SyncPhaseMode_MaxAcc := SyncModeCtrl.SyncPhase.MaxAcceleration;
        SyncPhaseMode_MaxDec := SyncModeCtrl.SyncPhase.MaxDeceleration;
        SyncPhaseMode_MaxJerk := SyncModeCtrl.SyncPhase.MaxJerk;
        SyncPhaseMode_MaxVelocity := SyncModeCtrl.SyncPhase.MaxVelocity;
        SyncPhaseMode_RatioNumerator := SyncModeCtrl.SyncPhase.OutputRevolution;
        SyncPhaseMode_RatioDenominator := SyncModeCtrl.SyncPhase.InputRevolution;
        SyncPhaseMode_SyncMode.GearInSyncMode := E_GearInSyncMode.GEARINSYNCMODE_POSITIONBASED;
        SyncPhaseMode_Enable := TRUE;
        AdminStatus.CmdDone := SyncPhaseControl.InSync;
    400:
        SyncPhaseMode_RealMasterPos := SyncModeCtrl.SyncPhase.Master.NcToPlc.ActPos + 10;
        SyncPhaseMode_RealSlavePos := AdminCtrl.Axis.NcToPlc.ActPos + 10;
        SyncPhaseMode_Master REF= SyncModeCtrl.SyncPhase.Master;
        SyncPhaseMode_MasterSyncPos := SyncPhaseMode_RealMasterPos;
        SyncPhaseMode_SlaveSyncPos := SyncPhaseMode_RealSlavePos;
        SyncPhaseMode_MaxAcc := SyncModeCtrl.SyncPhase.MaxAcceleration;
        SyncPhaseMode_MaxDec := SyncModeCtrl.SyncPhase.MaxDeceleration;
        SyncPhaseMode_MaxJerk := SyncModeCtrl.SyncPhase.MaxJerk;
        SyncPhaseMode_MaxVelocity := SyncModeCtrl.SyncPhase.MaxVelocity;
        SyncPhaseMode_RatioNumerator := SyncModeCtrl.SyncPhase.OutputRevolution;
        SyncPhaseMode_RatioDenominator := SyncModeCtrl.SyncPhase.InputRevolution;
        SyncPhaseMode_SyncMode.GearInSyncMode := E_GearInSyncMode.GEARINSYNCMODE_POSITIONBASED;
        SyncPhaseMode_SyncMode.GearInSync_CheckMask_MaxAcc := TRUE;
        SyncPhaseMode_SyncMode.GearInSync_CheckMask_MaxDec := TRUE;
        SyncPhaseMode_SyncMode.GearInSync_CheckMask_MaxJerk := TRUE;
        SyncPhaseMode_SyncMode.GearInSync_CheckMask_MaxVelo := TRUE;
        SyncPhaseMode_Enable := TRUE;

        //AdminStatus.CmdDone                   := SyncPhaseControl.InSync;

        //SuperInposMode := E_SuperpositionMode.SUPERPOSITIONMODE_LENGTHREDUCTION_ADDITIVEMOTION;
        IF SyncPhaseControl.InSync THEN
            uiModeSyncPhaseState := 500;
        END_IF
    500:
        // Calculate Axes Gap
        //        IF ABS(SyncPhaseMode_MasterModuleRemainder - SyncPhaseMode_SlaveModuleRemainder) > 180.0 THEN
        //            AxesGap := 360 - ABS(SyncPhaseMode_MasterModuleRemainder - SyncPhaseMode_SlaveModuleRemainder);
        //        ELSE
        //            AxesGap := ABS(SyncPhaseMode_MasterModuleRemainder - SyncPhaseMode_SlaveModuleRemainder);
        //        END_IF
        AxesGap := (SyncPhaseMode_MasterModuleRemainder - SyncPhaseMode_SlaveModuleRemainder);
        // SuperInpos start
        SuperInposMode := E_SuperpositionMode.SUPERPOSITIONMODE_LENGTHREDUCTION_ADDITIVEMOTION;

        //        IF (AxesGap - SyncModeCtrl.SyncPhase.MasterSyncPos - SyncModeCtrl.SyncPhase.SlaveSyncPos) >= 0 THEN
        //            SuperInposDistance := AxesGap + (SyncModeCtrl.SyncPhase.MasterSyncPos + SyncModeCtrl.SyncPhase.SlaveSyncPos);
        //        ELSE
        //            SuperInposDistance := 360 + (AxesGap + SyncModeCtrl.SyncPhase.MasterSyncPos + SyncModeCtrl.SyncPhase.SlaveSyncPos);
        //        END_IF
        SuperInposDistance := AxesGap + SyncModeCtrl.SyncPhase.MasterSyncPos + SyncModeCtrl.SyncPhase.SlaveSyncPos;
        //SuperInposDistance := AxesGap + (SyncModeCtrl.SyncPhase.MasterSyncPos + SyncModeCtrl.SyncPhase.SlaveSyncPos);
        PhaseOffsetSuperInpos.Length := 36000;
        PhaseOffsetSuperInpos.Execute := TRUE;
        SyncPhaseMode_SyncVelocity := SyncModeCtrl.SyncPhase.SyncVelocity;
        SyncPhaseMode_SyncAcceleration := SyncModeCtrl.SyncPhase.SyncAcceleration;
        SyncPhaseMode_LastMasterSyncPos := SyncModeCtrl.SyncPhase.MasterSyncPos;
        SyncPhaseMode_LastSlaveSyncPos := SyncModeCtrl.SyncPhase.SlaveSyncPos;

        IF PhaseOffsetSuperInpos.Execute THEN
            LastSuperInposDistance := SuperInposDistance;
            uiModeSyncPhaseState := 600;
        END_IF
    600:
        IF PhaseOffsetSuperInpos.Error THEN
            ;
        ELSIF PhaseOffsetSuperInpos.Done THEN

            uiModeSyncPhaseState := 700;
        END_IF
    700:
        PhaseOffsetSuperInpos.Execute := FALSE;
        uiModeSyncPhaseState := 710;
    710:
        IF (SyncModeCtrl.SyncPhase.MasterSyncPos <> SyncPhaseMode_LastMasterSyncPos) OR
            (SyncModeCtrl.SyncPhase.SlaveSyncPos <> SyncPhaseMode_LastSlaveSyncPos) OR
			((ModuleGap - (SyncModeCtrl.SyncPhase.MasterSyncPos +SyncModeCtrl.SyncPhase.SlaveSyncPos)) > 0.2)
		 THEN
			uiModeSyncPhaseState := 720;
        END_IF
	720:
		AxesGap2 := (SyncModeCtrl.SyncPhase.Master.NcToPlc.ModuloSetPos - AdminCtrl.Axis.NcToPlc.ModuloSetPos);
		IF ABS(AxesGap2 - (SyncModeCtrl.SyncPhase.MasterSyncPos +SyncModeCtrl.SyncPhase.SlaveSyncPos)) <= 180 THEN
			SuperInposDistance := AxesGap2 - (SyncModeCtrl.SyncPhase.MasterSyncPos +SyncModeCtrl.SyncPhase.SlaveSyncPos);
		ELSE
			IF (AxesGap2 - (SyncModeCtrl.SyncPhase.MasterSyncPos +SyncModeCtrl.SyncPhase.SlaveSyncPos)) >= 0 THEN
				SuperInposDistance := AxesGap2 - (SyncModeCtrl.SyncPhase.MasterSyncPos +SyncModeCtrl.SyncPhase.SlaveSyncPos)-360;
			ELSE
				SuperInposDistance := AxesGap2 - (SyncModeCtrl.SyncPhase.MasterSyncPos +SyncModeCtrl.SyncPhase.SlaveSyncPos)+360;
			END_IF
		END_IF
		
		//SuperInposDistance := AxesGap2 - (SyncModeCtrl.SyncPhase.MasterSyncPos +SyncModeCtrl.SyncPhase.SlaveSyncPos);
		
		PhaseOffsetSuperInpos.Length := 36000;
		PhaseOffsetSuperInpos.Execute := TRUE;
		uiModeSyncPhaseState := 730;
	730:
		IF PhaseOffsetSuperInpos.Error THEN
            ;
        ELSIF PhaseOffsetSuperInpos.Done THEN
			SyncPhaseMode_LastMasterSyncPos := SyncModeCtrl.SyncPhase.MasterSyncPos;
			SyncPhaseMode_LastSlaveSyncPos := SyncModeCtrl.SyncPhase.SlaveSyncPos;
            uiModeSyncPhaseState := 700;
        END_IF

END_CASE
END_ACTION

ACTION A08_ModeSyncVel:
IF NOT __ISVALIDREF(AdminCtrl) THEN
    RETURN;
END_IF

IF AdminCtrl._OpMode.en <> ModeSyncVel THEN
    SyncVelMode_Enable := FALSE;
    RETURN;
ELSIF AdminCtrl._OpMode.en <> LastOpMode THEN
    uiModeSyncVelState := 0;
    LastOpMode     := AdminCtrl._OpMode.en;
END_IF

CASE uiModeSyncVelState OF
    0:
        AdminStatus.CmdDone := FALSE;
        ClearAxisStatusBits();
        uiModeSyncVelState := 10;
    10:
        AdminStatus.ModeSyncVel := TRUE;
        AdminStatus._OpModeAck  := ModeSyncVel;

        IF AdminCtrl.Axis.Status.Disabled THEN
            uiModeSyncVelState := 100;
        ELSE
            uiModeSyncVelState := 200;
        END_IF
    100:
        // Power off -> Power On
        PowerOn(Direction := E_AxisDirection.Both);

        IF PowerControl.Status THEN
            uiModeSyncVelState := 200;
        END_IF
    200:
        SyncVelMode_Acc              := SyncModeCtrl.SyncVel.Acceleration;
        SyncVelMode_Dec              := SyncModeCtrl.SyncVel.Deceleration;
        SyncVelMode_Jerk             := SyncModeCtrl.SyncVel.Jerk;
        SyncVelMode_RatioNumerator   := SyncModeCtrl.SyncVel.OutputRevolution;
        SyncVelMode_RatioDenominator := SyncModeCtrl.SyncVel.InputRevolution;
		SyncVelMode_SyncMode.GearInSyncMode := E_GearInSyncMode.GEARINSYNCMODE_POSITIONBASED;
        //SyncVelMode_GearRatio := (SyncModeCtrl.SyncVel.OutputRevolution / SyncModeCtrl.SyncVel.InputRevolution) + SyncModeCtrl.SyncVel.FineAdjust;
        SyncVelMode_Master  REF= SyncModeCtrl.SyncVel.Master;
        SyncVelMode_Enable  := TRUE;
        AdminStatus.CmdDone := SyncVelControl.InSync;

END_CASE
END_ACTION

ACTION A09_ModeSyncCam:
(* ModeSyncCam is a mode that uses actions predefined with the Cam Design Tool. 
Once the cam profile is configured, it cannot be modified online, 
nor can it be changed via the PLC program.
*)
END_ACTION

ACTION A10_ModeSyncProfile:
IF NOT __ISVALIDREF(AdminCtrl) THEN
    RETURN;
END_IF

IF AdminCtrl._OpMode.en <> ModeSyncProfile THEN
    RETURN;
ELSIF AdminCtrl._OpMode.en <> LastOpMode THEN
    uiModeSyncProfile := 0;
    LastOpMode             := AdminCtrl._OpMode.en;
END_IF

CASE uiModeSyncProfile OF
	0:
        AdminStatus.CmdDone := FALSE;
        ClearAxisStatusBits();
		CamSelector.Execute := FALSE;
		CamInControl.Execute := FALSE;
        uiModeSyncProfile := 10;
    10:
        AdminStatus.ModeSyncProfile := TRUE;
        AdminStatus._OpModeAck  := ModeSyncProfile;

        IF AdminCtrl.Axis.Status.Disabled AND NOT AxisPowerON THEN
            uiModeSyncProfile := 100;
        ELSIF AdminCtrl.Axis.Status.Disabled AND AxisPowerON THEN
            PowerOFF();
			IF NOT AdminStatus.Active THEN
			uiModeSyncProfile := 200;
			END_IF
		ELSE
			uiModeSyncProfile := 200;
		END_IF
    100:
        // Power off -> Power On
        PowerOn(Direction := E_AxisDirection.Both);

        IF PowerControl.Status THEN
            uiModeSyncProfile := 3000; // JUMP TO NO OFFSET 
        END_IF
	200:
		// Move to CamIn Position
		IF AdminCtrl.PositionType = E_PositionType.Linear THEN
			uiModeSyncProfile := 3000;
		ELSIF AdminCtrl.PositionType = E_PositionType.Modulo THEN
			uiModeSyncProfile := 3000;
		END_IF
	1000:
		// move to linear offset position
	2000:
		// move to modulo offset position
	
	3000:
		// Select Cam profile
		SyncProfileMode_Master REF= SyncModeCtrl.SyncProfile.MasterAxis;
		SyncProfileMode_Periodic := SyncModeCtrl.SyncProfile.Periodic;
		SyncProfileMode_ProfileNum := SyncModeCtrl.SyncProfile.ProfileNum;
		SyncProfileMode_CamID := arCamID[SyncProfileMode_ProfileNum];
		SyncProfileMode_MasterOffset := SyncModeCtrl.SyncProfile.MasterOffset;
		SyncProfileMode_SlaveOffset := SyncModeCtrl.SyncProfile.SlaveOffset;
		SyncProfileMode_SyncType := SyncModeCtrl.SyncProfile.SyncType;
		SyncProfileOption.ActivationMode := MC_CAMACTIVATION_NEXTCYCLE;
		SyncProfileOption.InterpolationType :=MC_INTERPOLATIONTYPE_LINEAR;
		SyncProfileOption.MasterScalingMode := MC_CAMSCALING_USERDEFINED;
		SyncProfileOption.SlaveScalingMode := MC_CAMSCALING_AUTOOFFSET;
		
		CamSelector.Execute := TRUE;
		IF CamSelector.Error THEN
			DiagStatus.Error := TRUE;
			DiagStatus.ErrorID := CamSelector.ErrorID;
			DiagStatus.ErrorMsg := 'Cam select faild';
		ELSIF CamSelector.Done THEN
			uiModeSyncProfile := 3100;
		END_IF
	3100:
		// Cam In
		CamInControl.Execute := TRUE;
		IF CamInControl.Error THEN
			DiagStatus.Error := TRUE;
			DiagStatus.ErrorID := CamInControl.ErrorID;
			DiagStatus.ErrorMsg := 'Cam In faild';
		ELSIF CamInControl.InSync THEN
			AdminStatus.CmdDone := TRUE;
			uiModeSyncProfile := 9900;
		END_IF
	9900:
		// Wait command
END_CASE
END_ACTION

ACTION A11_ModeTorque:

END_ACTION

ACTION A12_ModeFlexProfile:
IF NOT __ISVALIDREF(AdminCtrl) THEN
    RETURN;
END_IF

IF AdminCtrl._OpMode.en <> ModeFlexProfile THEN
    RETURN;
ELSIF AdminCtrl._OpMode.en <> LastOpMode THEN
    uiModeFlexProfileState := 0;
    LastOpMode             := AdminCtrl._OpMode.en;
END_IF

CASE uiModeFlexProfileState OF
    0:
        AdminStatus.CmdDone := FALSE;
        ClearAxisStatusBits();
        uiModeFlexProfileState := 10;
    10:
        AdminStatus.ModePosAbs := TRUE;
        AdminStatus._OpModeAck := ModePosAbs;
        PosAbsMode_Execute     := FALSE;

        IF AdminCtrl.Axis.Status.Disabled THEN
            uiModeFlexProfileState := 100;
        ELSE
            uiModeFlexProfileState := 200;
        END_IF
    100:
        // Power off -> Power On
        PowerOn(Direction := E_AxisDirection.Both);

        IF PowerControl.Status THEN
            uiModeFlexProfileState := 200;
        END_IF
    200:
        // Move Master and Slave to Target position
        IF AdminCtrl.PositionType = E_PositionType.Linear THEN
            PosAbsMode_Position := SyncModeCtrl.SyncPhase.SlaveSyncPos;
            PosAbsMode_Velocity := SyncModeCtrl.SyncPhase.MaxVelocity;
            PosAbsMode_Acc      := SyncModeCtrl.SyncPhase.MaxAcceleration;
            PosAbsMode_Dec      := SyncModeCtrl.SyncPhase.MaxDeceleration;
            PosAbsMode_Jerk     := SyncModeCtrl.SyncPhase.MaxJerk;
            PosAbsMode_Execute  := TRUE;
        ELSIF AdminCtrl.PositionType = E_PositionType.Modulo THEN
            PosAbsMode_Position_Modulo := LMOD(SyncModeCtrl.SyncPhase.SlaveSyncPos, 360);
            PosAbsMode_Velocity_Modulo := SyncModeCtrl.SyncPhase.MaxVelocity;
            PosAbsMode_Acc_Modulo      := SyncModeCtrl.SyncPhase.MaxAcceleration;
            PosAbsMode_Dec_Modulo      := SyncModeCtrl.SyncPhase.MaxDeceleration;
            PosAbsMode_Jerk_Modulo     := SyncModeCtrl.SyncPhase.MaxJerk;
            PosAbsMode_Exectue_Modulo  := TRUE;
        END_IF

        CASE AdminCtrl.PositionType OF
            E_PositionType.Linear:
                IF MoveAbsControl.Done THEN
                    uiModeFlexProfileState := 300;
				ELSIF MoveAbsControl.Error THEN
					;
                END_IF
            E_PositionType.Modulo:
                IF MoveModuleControl.Done THEN
                    uiModeFlexProfileState := 300;
				ELSIF MoveModuleControl.Error THEN
					;
                END_IF
        END_CASE
	300:
		//
END_CASE
END_ACTION

ACTION A13_ModeStopping:

END_ACTION

ACTION A14_ModeCoordinated:
//IF NOT __ISVALIDREF(AdminCtrl) THEN
//	RETURN;
//END_IF

//IF (NcToPlc_gb.GrpId = 0) THEN
//	RETURN;
//END_IF
//IF AdminCtrl._OpMode.en <> ModeCoordinated THEN
//	RETURN;
//ELSIF AdminCtrl._OpMode.en <> LastOpMode THEN
//	uiModeCoordinatedState := 0;
//	LastOpMode := AdminCtrl._OpMode.en;
//END_IF

//CASE uiModeCoordinatedState OF 
//	0 : 
//		// Check Axis Status
//		IF AdminCtrl.Axis.Status.Disabled THEN
//			uiModeCoordinatedState := 100;
//		ELSE
//			uiModeCoordinatedState := 200;
//		END_IF
//	100:
//		// Power off -> Power On
//		PowerOn(Direction:= E_AxisDirection.Both);
//		IF PowerControl.Status THEN
//			uiModeCoordinatedState := 200;
//		END_IF
//	200:
//		IF ( AdminCtrl.Axis.Status.StandStill AND AdminCtrl.Axis.Status.NotMoving) THEN
//			uiModeCoordinatedState := 9000;
//		ELSE
//			uiModeCoordinatedState := 300;
//		END_IF
//	300:
//		// Stop Axis
//		AxisStop := TRUE;
//		AxisStop_Dec := AdminCtrl.StopDeceleration;
//		IF StopControl.Done THEN
//			uiModeCoordinatedState := 400;
//		END_IF
//	400:
//		AxisStop := FALSE;
//		AdminCtrl.ClearError := TRUE;
//		IF ResetControl.Done THEN
//			uiModeCoordinatedState := 500;
//		END_IF
//	500:
//		AdminCtrl.ClearError := FALSE;
//		ClearAxisStatusBits();
//		uiModeCoordinatedState := 9000;
//	9000:
//		// Setting Axis Status
//		AdminStatus.CmdDone := TRUE;
//		AdminStatus.ModeCoordinated := TRUE;
//		AdminStatus._OpModeAck := ModeCoordinated;
//		uiModeCoordinatedState := 10000;
//	10000:
//		// Wait command
//END_CASE
END_ACTION

ACTION A15_ModeInterrupted:

END_ACTION

ACTION A16_ModeExternalFB:

END_ACTION

ACTION A17_ModeCyclicPosition:

END_ACTION

ACTION A18_ModeCyclicVelocity:

END_ACTION

ACTION A19_ModeCyclicTorque:

END_ACTION

ACTION A80_AxisParaHandle:
(* ----- Axis Parameter -----*)

IF NOT bInitializePosBiasDone THEN
	bReadAxisPara:=TRUE;
END_IF

(* Read *)
IF bReadAxisPara THEN
	
	(* User defined path exists *)
	IF sAxisParaFolderPath <> '' THEN
		sTempString:=CONCAT(sAxisParaFolderPath,'\AxisParameter_');
		sTempString2:=CONCAT(TO_STRING(AdminCtrl.Axis.NcToPlc.AxisId),'.json');
		fbAxisParaHandler.sFilePath := CONCAT(sTempString, sTempString2);
	ELSE
		(* Default File path *)
		IF eOsType = E_OS_Type.WinCE THEN
			sTempString	:='\Hard Disk\TwinCAT\3.1\Boot\AxisParameter_';
			sTempString2:=CONCAT(TO_STRING(AdminCtrl.Axis.NcToPlc.AxisId),'.json');
			fbAxisParaHandler.sFilePath := CONCAT(sTempString, sTempString2);
		ELSIF eOsType = E_OS_Type.Windows  THEN
			sTempString	:='C:\TwinCAT\3.1\Boot\AxisParameter_';
			sTempString2:=CONCAT(TO_STRING(AdminCtrl.Axis.NcToPlc.AxisId),'.json');
			fbAxisParaHandler.sFilePath := CONCAT(sTempString, sTempString2);
		END_IF
	END_IF
	
	
	fbAxisParaHandler.eAction 	:= E_JsonHandlerAction.READ;
	fbAxisParaHandler.pData 	:= ADR(refAxisPara);
	fbAxisParaHandler.nData 	:= SIZEOF(refAxisPara);
	
	fbAxisParaHandler.xExecute	:=TRUE;
	
	IF fbAxisParaHandler.xDone THEN
		
		bReadAxisPara	:=FALSE;
		
		bInitializePosBiasDone	:=TRUE;
		
		fbAxisParaHandler.xExecute	:=FALSE;
		
	ELSIF fbAxisParaHandler.iErrorId = 9900 THEN(* File Not Exist *)
		
		(* When machine first time setup,there's no parameter file *)
		(* so see it as Init Done*) 
		bReadAxisPara	:=FALSE;
		bInitializePosBiasDone	:=TRUE;
		
		fbAxisParaHandler.xExecute	:=FALSE;
		
	END_IF
END_IF

(* -----FB Refresh----- *)
fbAxisParaHandler();
END_ACTION

ACTION A90_Cyclic:
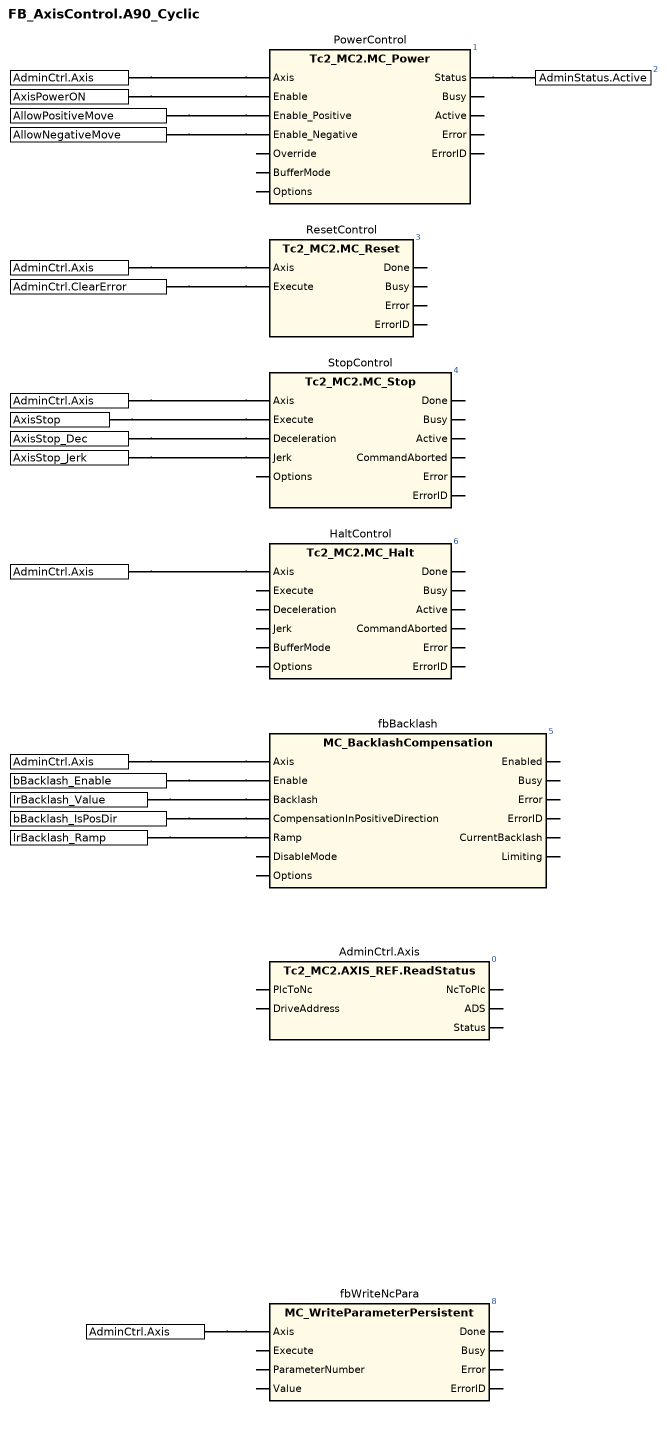
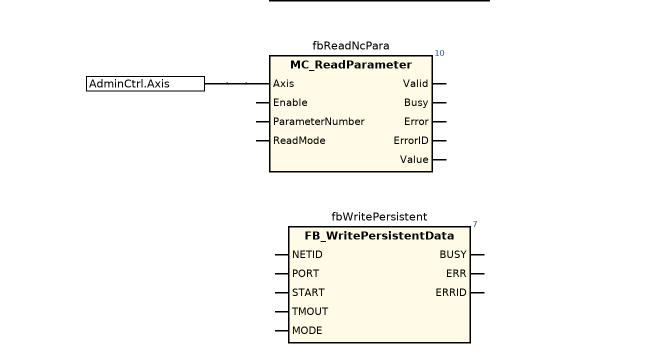
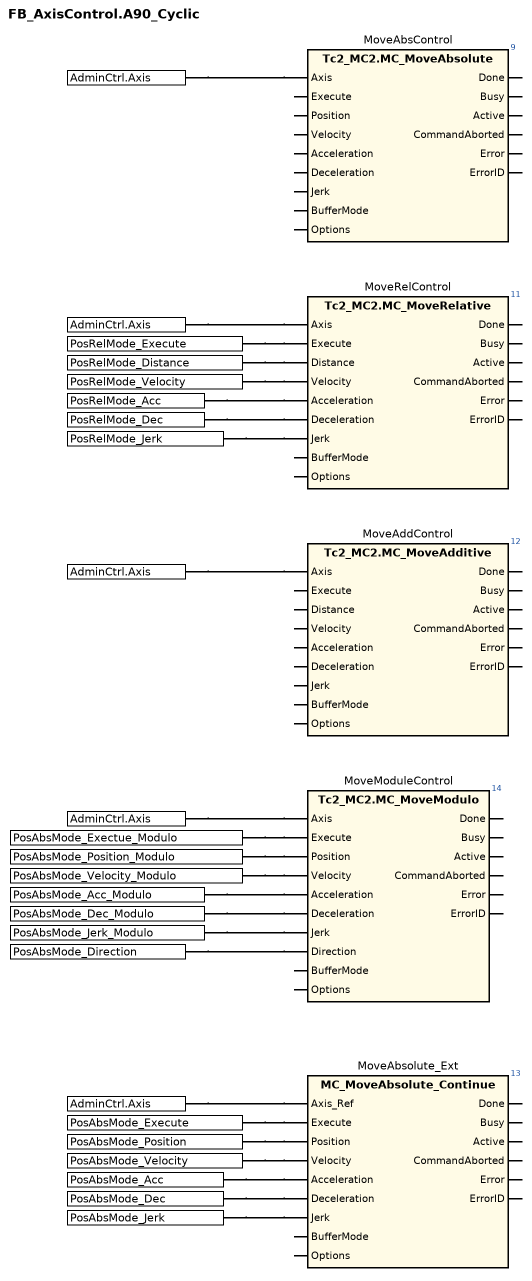
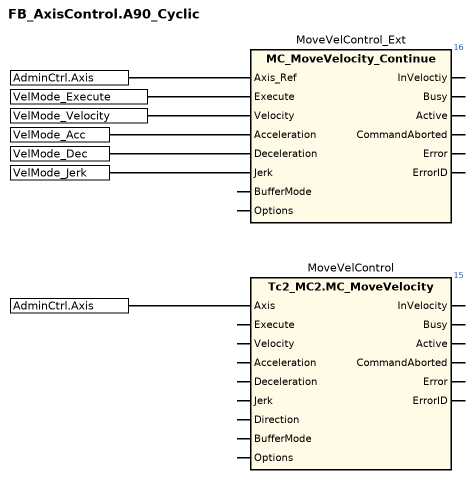
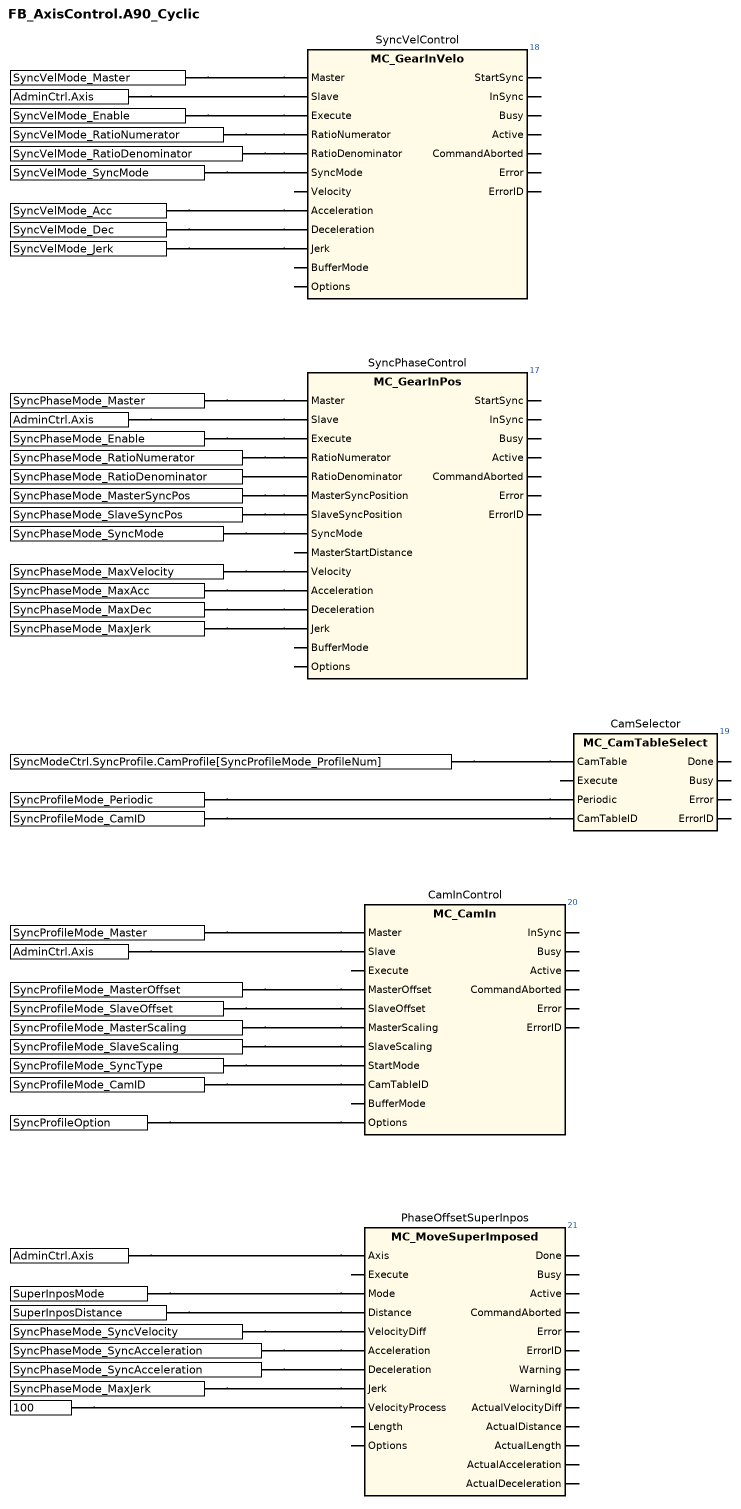
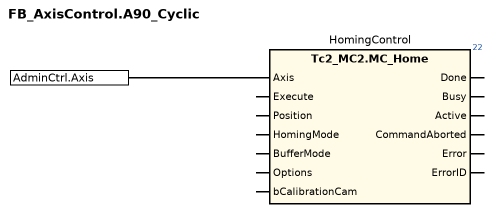
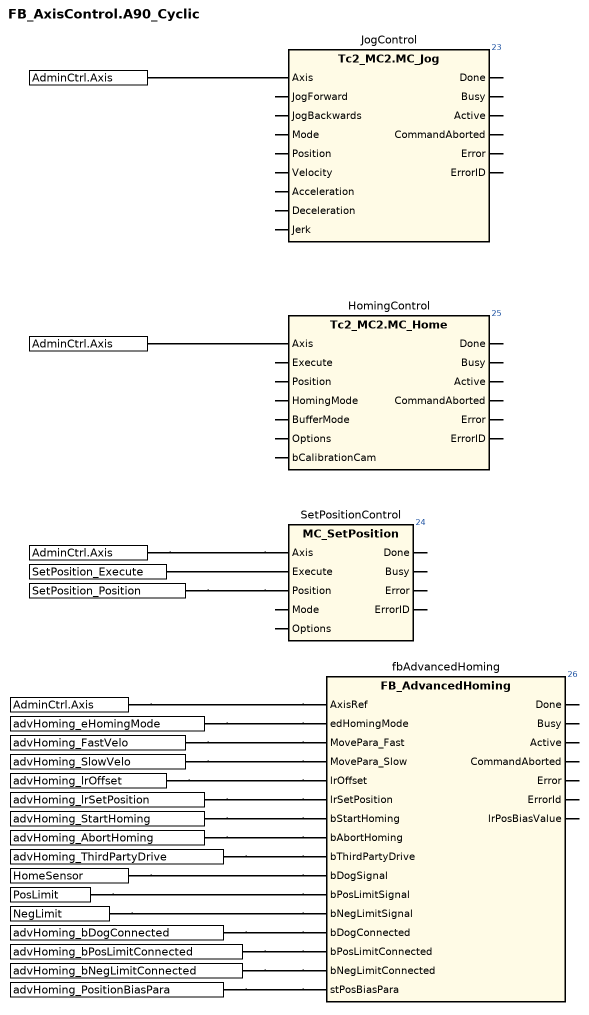
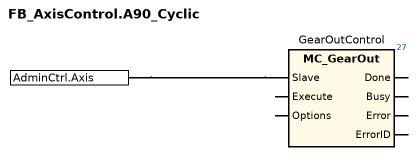
AdminCtrl.Axis.ReadStatus(); // Tc2_MC2.AXIS_REF.ReadStatus
PowerControl(
    Axis := AdminCtrl.Axis,
    Enable := AxisPowerON,
    Enable_Positive := AllowPositiveMove,
    Enable_Negative := AllowNegativeMove); // Tc2_MC2.MC_Power
AdminStatus.Active := PowerControl.Status;
ResetControl(Axis := AdminCtrl.Axis, Execute := AdminCtrl.ClearError); // Tc2_MC2.MC_Reset
StopControl(Axis := AdminCtrl.Axis, Execute := AxisStop, Deceleration := AxisStop_Dec, Jerk := AxisStop_Jerk); // Tc2_MC2.MC_Stop
fbBacklash(
    Axis := AdminCtrl.Axis,
    Enable := bBacklash_Enable,
    Backlash := lrBacklash_Value,
    CompensationInPositiveDirection := bBacklash_IsPosDir,
    Ramp := lrBacklash_Ramp); // MC_BacklashCompensation
HaltControl(Axis := AdminCtrl.Axis); // Tc2_MC2.MC_Halt
fbWritePersistent(); // FB_WritePersistentData
fbWriteNcPara(Axis := AdminCtrl.Axis); // MC_WriteParameterPersistent
MoveAbsControl(Axis := AdminCtrl.Axis); // Tc2_MC2.MC_MoveAbsolute
fbReadNcPara(Axis := AdminCtrl.Axis); // MC_ReadParameter
MoveRelControl(
    Axis := AdminCtrl.Axis,
    Execute := PosRelMode_Execute,
    Distance := PosRelMode_Distance,
    Velocity := PosRelMode_Velocity,
    Acceleration := PosRelMode_Acc,
    Deceleration := PosRelMode_Dec,
    Jerk := PosRelMode_Jerk); // Tc2_MC2.MC_MoveRelative
MoveAddControl(Axis := AdminCtrl.Axis); // Tc2_MC2.MC_MoveAdditive
MoveAbsolute_Ext(
    Axis_Ref := AdminCtrl.Axis,
    Execute := PosAbsMode_Execute,
    Position := PosAbsMode_Position,
    Velocity := PosAbsMode_Velocity,
    Acceleration := PosAbsMode_Acc,
    Deceleration := PosAbsMode_Dec,
    Jerk := PosAbsMode_Jerk); // MC_MoveAbsolute_Continue
MoveModuleControl(
    Axis := AdminCtrl.Axis,
    Execute := PosAbsMode_Exectue_Modulo,
    Position := PosAbsMode_Position_Modulo,
    Velocity := PosAbsMode_Velocity_Modulo,
    Acceleration := PosAbsMode_Acc_Modulo,
    Deceleration := PosAbsMode_Dec_Modulo,
    Jerk := PosAbsMode_Jerk_Modulo,
    Direction := PosAbsMode_Direction); // Tc2_MC2.MC_MoveModulo
MoveVelControl(Axis := AdminCtrl.Axis); // Tc2_MC2.MC_MoveVelocity
MoveVelControl_Ext(
    Axis_Ref := AdminCtrl.Axis,
    Execute := VelMode_Execute,
    Velocity := VelMode_Velocity,
    Acceleration := VelMode_Acc,
    Deceleration := VelMode_Dec,
    Jerk := VelMode_Jerk); // MC_MoveVelocity_Continue
SyncPhaseControl(
    Master := SyncPhaseMode_Master,
    Slave := AdminCtrl.Axis,
    Execute := SyncPhaseMode_Enable,
    RatioNumerator := SyncPhaseMode_RatioNumerator,
    RatioDenominator := SyncPhaseMode_RatioDenominator,
    MasterSyncPosition := SyncPhaseMode_MasterSyncPos,
    SlaveSyncPosition := SyncPhaseMode_SlaveSyncPos,
    SyncMode := SyncPhaseMode_SyncMode,
    Velocity := SyncPhaseMode_MaxVelocity,
    Acceleration := SyncPhaseMode_MaxAcc,
    Deceleration := SyncPhaseMode_MaxDec,
    Jerk := SyncPhaseMode_MaxJerk); // MC_GearInPos
SyncVelControl(
    Master := SyncVelMode_Master,
    Slave := AdminCtrl.Axis,
    Execute := SyncVelMode_Enable,
    RatioNumerator := SyncVelMode_RatioNumerator,
    RatioDenominator := SyncVelMode_RatioDenominator,
    SyncMode := SyncVelMode_SyncMode,
    Acceleration := SyncVelMode_Acc,
    Deceleration := SyncVelMode_Dec,
    Jerk := SyncVelMode_Jerk); // MC_GearInVelo
CamSelector(
    CamTable := SyncModeCtrl.SyncProfile.CamProfile[SyncProfileMode_ProfileNum],
    Periodic := SyncProfileMode_Periodic,
    CamTableID := SyncProfileMode_CamID); // MC_CamTableSelect
CamInControl(
    Master := SyncProfileMode_Master,
    Slave := AdminCtrl.Axis,
    MasterOffset := SyncProfileMode_MasterOffset,
    SlaveOffset := SyncProfileMode_SlaveOffset,
    MasterScaling := SyncProfileMode_MasterScaling,
    SlaveScaling := SyncProfileMode_SlaveScaling,
    StartMode := SyncProfileMode_SyncType,
    CamTableID := SyncProfileMode_CamID,
    Options := SyncProfileOption); // MC_CamIn
PhaseOffsetSuperInpos(
    Axis := AdminCtrl.Axis,
    Mode := SuperInposMode,
    Distance := SuperInposDistance,
    VelocityDiff := SyncPhaseMode_SyncVelocity,
    Acceleration := SyncPhaseMode_SyncAcceleration,
    Deceleration := SyncPhaseMode_SyncAcceleration,
    Jerk := SyncPhaseMode_MaxJerk,
    VelocityProcess := 100); // MC_MoveSuperImposed
HomingControl(Axis := AdminCtrl.Axis); // Tc2_MC2.MC_Home
JogControl(Axis := AdminCtrl.Axis); // Tc2_MC2.MC_Jog
SetPositionControl(Axis := AdminCtrl.Axis, Execute := SetPosition_Execute, Position := SetPosition_Position); // MC_SetPosition
HomingControl(Axis := AdminCtrl.Axis); // Tc2_MC2.MC_Home
fbAdvancedHoming(
    AxisRef := AdminCtrl.Axis,
    edHomingMode := advHoming_eHomingMode,
    MovePara_Fast := advHoming_FastVelo,
    MovePara_Slow := advHoming_SlowVelo,
    lrOffset := advHoming_lrOffset,
    lrSetPosition := advHoming_lrSetPosition,
    bStartHoming := advHoming_StartHoming,
    bAbortHoming := advHoming_AbortHoming,
    bThirdPartyDrive := advHoming_ThirdPartyDrive,
    bDogSignal := HomeSensor,
    bPosLimitSignal := PosLimit,
    bNegLimitSignal := NegLimit,
    bDogConnected := advHoming_bDogConnected,
    bPosLimitConnected := advHoming_bPosLimitConnected,
    bNegLimitConnected := advHoming_bNegLimitConnected,
    stPosBiasPara := advHoming_PositionBiasPara); // FB_AdvancedHoming
GearOutControl(Slave := AdminCtrl.Axis); // MC_GearOut
END_ACTION

METHOD M_InitExtension
VAR_INPUT
	Index : UDINT;
END_VAR
//=============================================================//
//Reference access											   //
//=============================================================//
AdminCtrl      REF= arAxisCtrl_gb[Index].Admin;
PosModeCtrl    REF= arAxisCtrl_gb[Index].PosMode;
VelModeCtrl    REF= arAxisCtrl_gb[Index].VelMode;
SyncModeCtrl   REF= arAxisCtrl_gb[Index].SyncMode;
TorqueModeCtrl REF= arAxisCtrl_gb[Index].TorqueMode;
SetupModeCtrl  REF= arAxisCtrl_gb[Index].SetupMode;

AdminStatus     REF= arAxisStatus_gb[Index].Admin;
DiagStatus      REF= arAxisStatus_gb[Index].Diag;
PosModeStatus   REF= arAxisStatus_gb[Index].PosMode;
VelModeStatus   REF= arAxisStatus_gb[Index].VelMode;
SyncModeStatus  REF= arAxisStatus_gb[Index].SyncMode;
SetupModeStatus REF= arAxisStatus_gb[Index].SetupMode;

////refNcPositionBias REF= arAxisBias_gb[Index];
refAxisPara 	 REF= arAxisPara_gb[Index];
fbAdvancedHoming.refAxisPara REF= refAxisPara;

//=============================================================//
//Memory Axis ID											   //
//=============================================================//
AxisID     := Index;
arCamID[1] := (4 * AxisID) - 4;
arCamID[2] := (4 * AxisID) - 3;
arCamID[3] := (4 * AxisID) - 2;
arCamID[4] := (4 * AxisID) - 1;

//=============================================================//
//Read Axis Address											   //
//=============================================================//
fbReadAxisAddress(
	Axis:= AdminCtrl.Axis, 
	Execute:= TRUE, 
	Done=> , 
	Busy=> , 
	Error=> , 
	ErrorID=> , 
	DriveAddress=> AdminStatus.DriverAddress);
END_METHOD

END_FUNCTION_BLOCK

// AxisInterface/LIB/AxisControl/MC_MoveVelocity_Continue
(* This Function block is used to switch velocity command 
*)
FUNCTION_BLOCK MC_MoveVelocity_Continue
VAR_INPUT
    Axis_Ref     : REFERENCE TO AXIS_REF;
    Execute      : BOOL;
    Velocity     : LREAL;
    Acceleration : LREAL;
    Deceleration : LREAL;
    Jerk         : LREAL;
    BufferMode   : MC_BufferMode:= MC_BufferMode.MC_Buffered;
    Options      : ST_MoveOptions;
END_VAR
VAR_OUTPUT
    InVeloctiy     : BOOL;
    Busy           : BOOL;
    Active         : BOOL;
    CommandAborted : BOOL;
    Error          : BOOL;
    ErrorID        : UDINT;
END_VAR
VAR
    fb_MoveVelocity_1st : Tc2_MC2.MC_MoveVelocity;
    fb_MoveVelocity_2nd : Tc2_MC2.MC_MoveVelocity;
	Velocity_Old : LREAL;
	Acceleration_Old : LREAL;
	Deceleration_Old : LREAL;
	Jerk_Old : LREAL;
	bNeedSwitch : BOOL;
	VelMode_Dir : MC_Direction;
	Velocity_CMD1 : BOOL;
	Velocity_CMD2 : BOOL;
	udiVelocityStep : UDINT;
	fbExecute_Rtrig :R_TRIG;
	fbExecute_Ftrig :F_TRIG;
END_VAR

fbExecute_Rtrig(CLK := Execute, Q =>);
fbExecute_Ftrig(CLK := Execute, Q =>);

IF fbExecute_Ftrig.Q THEN
    udiVelocityStep := 0;
END_IF

IF Velocity > 0 THEN
    VelMode_Dir := MC_Direction.MC_Positive_Direction;
ELSIF Velocity < 0 THEN
    VelMode_Dir := MC_Direction.MC_Negative_Direction;
END_IF

CASE udiVelocityStep OF
    0:
        Velocity_CMD1 := FALSE;
        Velocity_CMD2 := FALSE;
		
        IF Execute THEN
            udiVelocityStep := 10;
        END_IF
	10:
		IF Axis_Ref.Status.Coupled THEN
			BufferMode := MC_BufferMode.MC_Aborting;
			udiVelocityStep:=100;
		ELSE
			udiVelocityStep:=100;
		END_IF
    100:
        Velocity_CMD1 := TRUE;

        IF fb_MoveVelocity_1st.Busy THEN
            Velocity_Old     := Velocity;
            Acceleration_Old := Acceleration;
            Deceleration_Old := Deceleration;
            Jerk_Old         := Jerk;
            udiVelocityStep  := 200;
        END_IF
    200:
        // Wait command change
        IF (Velocity_Old <> Velocity) OR
            (Acceleration_Old <> Acceleration) OR
            (Deceleration_Old <> Deceleration) OR
            (Jerk_Old <> Jerk) THEN
			IF NOT Axis_Ref.Status.Coupled THEN
				BufferMode := MC_BufferMode.MC_Buffered;
			END_IF
            udiVelocityStep := 300;
        END_IF
    300:
        Velocity_CMD2 := TRUE;

        IF fb_MoveVelocity_2nd.Busy THEN
            Velocity_Old     := Velocity;
            Acceleration_Old := Acceleration;
            Deceleration_Old := Deceleration;
            Jerk_Old         := Jerk;
            udiVelocityStep := 400;
        END_IF

    400:
        Velocity_CMD1 := FALSE;

        IF NOT fb_MoveVelocity_1st.Busy THEN
            udiVelocityStep := 500;
        END_IF
    500:
        // Wait command change
        IF (Velocity_Old <> Velocity) OR
            (Acceleration_Old <> Acceleration) OR
            (Deceleration_Old <> Deceleration) OR
            (Jerk_Old <> Jerk) THEN
			IF NOT Axis_Ref.Status.Coupled THEN
				BufferMode := MC_BufferMode.MC_Buffered;
			END_IF
            udiVelocityStep := 600;
        END_IF
    600:
        Velocity_CMD1 := TRUE;

        IF fb_MoveVelocity_1st.Busy THEN
            Velocity_Old     := Velocity;
            Acceleration_Old := Acceleration;
            Deceleration_Old := Deceleration;
            Jerk_Old         := Jerk;
            udiVelocityStep := 700;
        END_IF
    700:
        Velocity_CMD2 := FALSE;

        IF NOT fb_MoveVelocity_2nd.Busy THEN
            udiVelocityStep := 800;
        END_IF
    800:
        // Wait command change
        IF (Velocity_Old <> Velocity) OR
            (Acceleration_Old <> Acceleration) OR
            (Deceleration_Old <> Deceleration) OR
            (Jerk_Old <> Jerk) THEN
			IF NOT Axis_Ref.Status.Coupled THEN
				BufferMode := MC_BufferMode.MC_Buffered;
			END_IF
            udiVelocityStep := 300;
        END_IF
END_CASE

fb_MoveVelocity_1st(Axis           := Axis_Ref,
                    Execute        := Velocity_CMD1,
                    Velocity       := ABS(Velocity),
                    Acceleration   := Acceleration,
                    Deceleration   := Deceleration,
                    Jerk           := Jerk,
                    Direction      := VelMode_Dir,
                    BufferMode     := BufferMode,
                    Options        :=,
                    InVelocity     =>,
                    Busy           =>,
                    Active         =>,
                    CommandAborted =>,
                    Error          =>,
                    ErrorID        =>);

fb_MoveVelocity_2nd(Axis           := Axis_Ref,
                    Execute        := Velocity_CMD2,
                    Velocity       := ABS(Velocity),
                    Acceleration   := Acceleration,
                    Deceleration   := Deceleration,
                    Jerk           := Jerk,
                    Direction      := VelMode_Dir,
                    BufferMode     := BufferMode,
                    Options        :=,
                    InVelocity     =>,
                    Busy           =>,
                    Active         =>,
                    CommandAborted =>,
                    Error          =>,
                    ErrorID        =>);

IF fb_MoveVelocity_1st.Busy THEN
    InVeloctiy     := fb_MoveVelocity_1st.InVelocity;
    Busy           := fb_MoveVelocity_1st.Busy;
    Active         := fb_MoveVelocity_1st.Active;
    CommandAborted := fb_MoveVelocity_1st.CommandAborted;
    Error          := fb_MoveVelocity_1st.Error;
    ErrorID        := fb_MoveVelocity_1st.ErrorID;
ELSIF fb_MoveVelocity_2nd.Busy THEN
    InVeloctiy     := fb_MoveVelocity_2nd.InVelocity;
    Busy           := fb_MoveVelocity_2nd.Busy;
    Active         := fb_MoveVelocity_2nd.Active;
    CommandAborted := fb_MoveVelocity_2nd.CommandAborted;
    Error          := fb_MoveVelocity_2nd.Error;
    ErrorID        := fb_MoveVelocity_2nd.ErrorID;
ELSE
    InVeloctiy     := FALSE;
    Busy           := FALSE;
    Active         := FALSE;
    CommandAborted := FALSE;
    Error          := FALSE;
    ErrorID        := 0;
END_IF

END_FUNCTION_BLOCK

// AxisInterface/LIB/AxisControl/MC_MoveAbsolute_Continue
FUNCTION_BLOCK MC_MoveAbsolute_Continue
VAR_INPUT
    Axis_Ref     : REFERENCE TO AXIS_REF;
    Execute      : BOOL;
    Position     : LREAL;
    Velocity     : LREAL;
    Acceleration : LREAL;
    Deceleration : LREAL;
    Jerk         : LREAL;
    BufferMode   : MC_BufferMode := MC_BufferMode.MC_Aborting;
    Options      : ST_MoveOptions;
END_VAR
VAR_OUTPUT
    Done           : BOOL;
    Busy           : BOOL;
    Active         : BOOL;
    CommandAborted : BOOL;
    Error          : BOOL;
    ErrorID        : UDINT;
END_VAR
VAR
    udiAbsoluteStep     : UDINT;
    fb_MoveAbsolute_1st : MC_MoveAbsolute;
    fb_MoveAbsolute_2nd : MC_MoveAbsolute;
    Position_Old        : LREAL;
    Velocity_Old        : LREAL;
    Acceleration_Old    : LREAL;
    Deceleration_Old    : LREAL;
    Jerk_Old            : LREAL;
    fbExecute_Rtrig     : R_TRIG;
    fbExecute_Ftrig     : F_TRIG;
    Absolute_CMD1       : BOOL;
    Absolute_CMD2       : BOOL;
END_VAR

fbExecute_Ftrig(CLK := Execute, Q =>);

IF fbExecute_Ftrig.Q THEN
    udiAbsoluteStep := 0;
END_IF

CASE udiAbsoluteStep OF
    0:
        Absolute_CMD1 := FALSE;
        Absolute_CMD2 := FALSE;

        IF Execute THEN
            udiAbsoluteStep := 100;
        END_IF
    100:
        Absolute_CMD1 := TRUE;

        IF fb_MoveAbsolute_1st.Busy OR fb_MoveAbsolute_1st.Done THEN
            Position_Old     := Position;
            Velocity_Old     := Velocity;
            Acceleration_Old := Acceleration;
            Deceleration_Old := Deceleration;
            Jerk_Old         := Jerk;
            udiAbsoluteStep  := 200;
        END_IF
    200:
        // Wait command change
        IF (Position_Old <> Position) OR
            (Velocity_Old <> Velocity) OR
            (Acceleration_Old <> Acceleration) OR
            (Deceleration_Old <> Deceleration) OR
            (Jerk_Old <> Jerk) THEN
            udiAbsoluteStep := 300;
        END_IF
    300:
        Absolute_CMD2 := TRUE;

        IF fb_MoveAbsolute_2nd.Busy OR fb_MoveAbsolute_2nd.Done THEN
            Position_Old     := Position;
            Velocity_Old     := Velocity;
            Acceleration_Old := Acceleration;
            Deceleration_Old := Deceleration;
            Jerk_Old         := Jerk;
            udiAbsoluteStep  := 400;
        END_IF
    400:
        Absolute_CMD1 := FALSE;

        IF NOT fb_MoveAbsolute_1st.Busy AND NOT fb_MoveAbsolute_1st.Done THEN
            udiAbsoluteStep := 500;
        END_IF
    500:
        // Wait command change
        IF (Position_Old <> Position) OR
            (Velocity_Old <> Velocity) OR
            (Acceleration_Old <> Acceleration) OR
            (Deceleration_Old <> Deceleration) OR
            (Jerk_Old <> Jerk) THEN
            udiAbsoluteStep := 600;
        END_IF
    600:
        Absolute_CMD1 := TRUE;

        IF fb_MoveAbsolute_1st.Busy OR fb_MoveAbsolute_1st.Done THEN
            Position_Old     := Position;
            Velocity_Old     := Velocity;
            Acceleration_Old := Acceleration;
            Deceleration_Old := Deceleration;
            Jerk_Old         := Jerk;
            udiAbsoluteStep  := 700;
        END_IF
    700:
        Absolute_CMD2 := FALSE;

        IF NOT fb_MoveAbsolute_2nd.Busy AND NOT fb_MoveAbsolute_2nd.Done THEN
            udiAbsoluteStep := 800;
        END_IF
    800:
        // Wait command change
        IF (Position_Old <> Position) OR
            (Velocity_Old <> Velocity) OR
            (Acceleration_Old <> Acceleration) OR
            (Deceleration_Old <> Deceleration) OR
            (Jerk_Old <> Jerk) THEN
            udiAbsoluteStep := 300;
        END_IF
END_CASE

fb_MoveAbsolute_1st(Axis           := Axis_Ref,
                    Execute        := Absolute_CMD1,
                    Position       := Position,
                    Velocity       := Velocity,
                    Acceleration   := Acceleration,
                    Deceleration   := Deceleration,
                    Jerk           := Jerk,
                    BufferMode     := BufferMode,
                    Options        := Options,
                    Done           =>,
                    Busy           =>,
                    Active         =>,
                    CommandAborted =>,
                    Error          =>,
                    ErrorID        =>);

fb_MoveAbsolute_2nd(Axis           := Axis_Ref,
                    Execute        := Absolute_CMD2,
                    Position       := Position,
                    Velocity       := Velocity,
                    Acceleration   := Acceleration,
                    Deceleration   := Deceleration,
                    Jerk           := Jerk,
                    BufferMode     := BufferMode,
                    Options        := Options,
                    Done           =>,
                    Busy           =>,
                    Active         =>,
                    CommandAborted =>,
                    Error          =>,
                    ErrorID        =>);

IF fb_MoveAbsolute_1st.Execute THEN
    Done           := fb_MoveAbsolute_1st.Done;
    Busy           := fb_MoveAbsolute_1st.Busy;
    Active         := fb_MoveAbsolute_1st.Active;
    CommandAborted := fb_MoveAbsolute_1st.CommandAborted;
    Error          := fb_MoveAbsolute_1st.Error;
    ErrorID        := fb_MoveAbsolute_1st.ErrorID;
ELSIF fb_MoveAbsolute_2nd.Execute THEN
    Done           := fb_MoveAbsolute_2nd.Done;
    Busy           := fb_MoveAbsolute_2nd.Busy;
    Active         := fb_MoveAbsolute_2nd.Active;
    CommandAborted := fb_MoveAbsolute_2nd.CommandAborted;
    Error          := fb_MoveAbsolute_2nd.Error;
    ErrorID        := fb_MoveAbsolute_2nd.ErrorID;
ELSE
    Done           := FALSE;
    Busy           := FALSE;
    Active         := FALSE;
    CommandAborted := FALSE;
    Error          := FALSE;
    ErrorID        := 0;
END_IF

END_FUNCTION_BLOCK

// AxisInterface/LIB/AxisControl/FB_AdvancedHoming
FUNCTION_BLOCK FB_AdvancedHoming
VAR_IN_OUT
    AxisRef : AXIS_REF;
END_VAR
VAR_INPUT
    edHomingMode        : E_HomingMode;
    MovePara_Fast       : ST_VelocityParameter := (Velocity := 10, Acc := 100, Dec := 100, Jerk := 1000); //Default High Speed
    MovePara_Slow       : ST_VelocityParameter := (Velocity := 1, Acc := 10, Dec := 10, Jerk := 100); //Default Low Speed
    MoveLimitation_Fast : ST_HomingLimitation;
    MoveLimitation_Slow : ST_HomingLimitation;

    lrOffset      : LREAL; //Distance by which the axis moves away from the current position.
    lrSetPosition : LREAL; //Position value to which the axis position is set to.

    bStartHoming     : BOOL;
    bAbortHoming     : BOOL;
    bThirdPartyDrive : BOOL;

    //Signal Handle
    bDogSignal : BOOL;
    //bZeroPulseSigal		:BOOL;
    bPosLimitSignal    : BOOL;
    bNegLimitSignal    : BOOL;
    bDogConnected      : BOOL;
    bPosLimitConnected : BOOL;
    bNegLimitConnected : BOOL;
    //Position Bias
    //refNcPositionBias 	: REFERENCE TO LREAL;//Reference to arAxisBias_gb
    stPosBiasPara : ST_PositionBiasParameter;
    refAxisPara   : REFERENCE TO ST_AXIS_Parameter;
END_VAR
VAR_OUTPUT
    Done           : BOOL; // TRUE : when the absolute phase shift is established.
    Busy           : BOOL; // TRUE as soon as the command is started with Execute and as long as the phase shift occurs.
    Active         : BOOL; // Indicates that the command is executed. 
    CommandAborted : BOOL; // TRUE if the command could not be executed completely. 
    Error          : BOOL; // TRUE, if an error occurs.
    ErrorId        : UDINT;
    lrPosBiasValue : LREAL; //  Position Bias need to be set
END_VAR
VAR
    //-----FBs-----
    //Step Function
    fbStepAbsoluteSwitchDetection : MC_StepAbsoluteSwitchDetection;
    fbStepAbsoluteSwitch          : MC_StepAbsoluteSwitch;
    fbStepLimitSwitchDetection    : MC_StepLimitSwitchDetection;
    fbStepLimitSwitch             : MC_StepLimitSwitch;
    fbStepReferencePulse          : MC_StepReferencePulse;
    fbStepReferencePulseDetection : MC_StepReferencePulseDetection;
    fbMoveAbs                     : MC_MoveAbsolute;
    //Finanlizing Function
    fbFinishHoming : MC_FinishHoming;
    fbHomeDirect   : MC_HomeDirect;
    fbAbortHoming  : MC_AbortHoming;

    //NC Parameters
    fbReadParameter : MC_ReadParameter;

    //-----Parameter-----
    Parameter : MC_HomingParameter;
    Options4  : ST_Home_Options4;
    Options2  : ST_Home_Options2;

    //-----Signals-----
    PosLimitSwitchSignal : MC_Ref_Signal_Ref;
    NegLimitSwitchSignal : MC_Ref_Signal_Ref;
    DogSignal            : MC_Ref_Signal_Ref;
    ZeroSwitchSignal     : MC_Ref_Signal_Ref;

END_VAR
VAR
    //Vars
    uiCurrentCmdNo      : UINT;
    uiCommandDoneNum    : UINT;
    eHome_ActionType    : E_HomingActionType;
    stAdvHomePara_Local : ST_AdvancedHoming_Parameter; //Use to Executing Homing Procedure, this Var will get from stAdvHomePara_Set before Executing
    stAdvHomePara_Set   : ST_AdvancedHoming_Parameter; //Use to Set Command List content to this Var
    stAdvHomePara_Clear : ST_AdvancedHoming_Parameter; //Use to Clear Command List content before set new Command List

    //Action Trigger
    rTrig_Start : R_TRIG;
    fTrig_Start : F_TRIG;
    rTrig_Abort : R_TRIG;
    fTrig_Abort : F_TRIG;

    //Step
    iStep_Homing         : INT;
    iStep_StepFunc       : INT;
    iStep_FinalizingFunc : INT;
    iStep_ParaSetting    : INT;

    uiStepFuncErrorId : UDINT;
END_VAR
VAR
    {attribute 'hide'}
    bSimuMode : BOOL := FALSE;
END_VAR

//FB Refresh
A_CyclicUpdate();

//Action Trigger
A_ActionTrigger();

CASE iStep_Homing OF
	0:
	(*-----Executing-----*)
	100://Check Step
	
		//Check if Command List Correct
		IF stAdvHomePara_Set.uiCommandNum > 0 
		AND edHomingMode <> E_HomingMode.notDefined THEN
		
